Yaskawa INFORM job: A_ROOF_SIDE_0617_2_PAINT_58.JBI

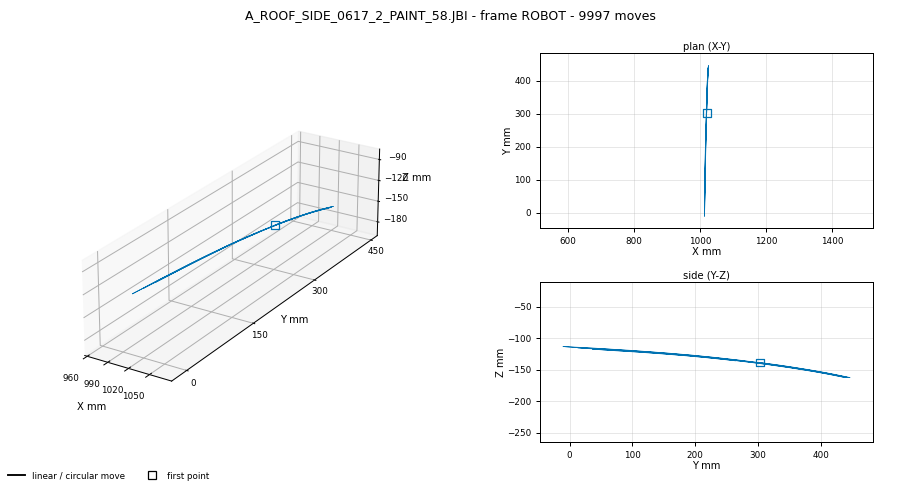
[picture p0: tool path of A_ROOF_SIDE_0617_2_PAINT_58.JBI in frame ROBOT, 9997 of 9997 moves have a stored position in this frame; points joined in program order, loops and branches not executed]
/JOB
//NAME A_ROOF_SIDE_0617_2_PAINT58
//POS
///NPOS 9997,0,0,0,0,0
///TOOL 1
///USER 0
///POSTYPE ROBOT
///RECTAN
///RCONF 1,0,0,0,0,0,0,0,0,0,0,0,0,0,0,0,0,0,0,0,0,0,0,0
C00000=1019.451,302.645,-138.347,170.187,50.132,159.718
C00001=1019.458,302.892,-138.379,170.193,50.128,159.718
C00002=1019.464,303.141,-138.411,170.199,50.124,159.718
C00003=1019.471,303.388,-138.443,170.204,50.121,159.718
C00004=1019.478,303.636,-138.476,170.209,50.117,159.718
C00005=1019.484,303.884,-138.508,170.215,50.113,159.718
C00006=1019.491,304.131,-138.540,170.220,50.110,159.718
C00007=1019.498,304.379,-138.573,170.227,50.106,159.719
C00008=1019.504,304.627,-138.604,170.232,50.103,159.719
C00009=1019.511,304.875,-138.637,170.237,50.099,159.719
C00010=1019.517,305.122,-138.670,170.243,50.095,159.719
C00011=1019.524,305.370,-138.701,170.248,50.092,159.719
C00012=1019.530,305.618,-138.734,170.255,50.088,159.719
C00013=1019.538,305.866,-138.767,170.260,50.085,159.719
C00014=1019.544,306.113,-138.799,170.265,50.082,159.719
C00015=1019.550,306.362,-138.831,170.271,50.077,159.719
C00016=1019.557,306.609,-138.864,170.276,50.074,159.719
C00017=1019.564,306.857,-138.897,170.283,50.070,159.720
C00018=1019.570,307.101,-138.929,170.288,50.067,159.720
C00019=1019.576,307.344,-138.960,170.293,50.064,159.720
C00020=1019.583,307.587,-138.992,170.299,50.060,159.720
C00021=1019.590,307.830,-139.025,170.305,50.057,159.720
C00022=1019.596,308.074,-139.056,170.310,50.053,159.720
C00023=1019.604,308.318,-139.089,170.316,50.050,159.720
C00024=1019.610,308.562,-139.121,170.322,50.046,159.720
C00025=1019.617,308.805,-139.152,170.327,50.043,159.721
C00026=1019.624,309.052,-139.185,170.333,50.039,159.721
C00027=1019.630,309.300,-139.217,170.338,50.036,159.721
C00028=1019.637,309.548,-139.250,170.345,50.033,159.721
C00029=1019.644,309.796,-139.283,170.350,50.029,159.721
C00030=1019.650,310.043,-139.315,170.356,50.026,159.721
C00031=1019.658,310.291,-139.349,170.362,50.023,159.722
C00032=1019.663,310.539,-139.382,170.367,50.020,159.722
C00033=1019.669,310.786,-139.415,170.373,50.016,159.722
C00034=1019.677,311.034,-139.449,170.379,50.013,159.722
C00035=1019.683,311.282,-139.482,170.384,50.010,159.722
C00036=1019.689,311.529,-139.515,170.391,50.007,159.723
C00037=1019.696,311.777,-139.549,170.396,50.004,159.723
C00038=1019.702,312.025,-139.582,170.402,50.000,159.723
C00039=1019.709,312.272,-139.615,170.408,49.997,159.723
C00040=1019.715,312.520,-139.648,170.414,49.994,159.723
C00041=1019.721,312.767,-139.682,170.419,49.991,159.724
C00042=1019.728,313.015,-139.715,170.425,49.988,159.724
C00043=1019.735,313.263,-139.749,170.431,49.984,159.724
C00044=1019.741,313.510,-139.782,170.437,49.981,159.724
C00045=1019.748,313.758,-139.816,170.443,49.978,159.724
C00046=1019.754,314.006,-139.849,170.448,49.976,159.725
C00047=1019.761,314.254,-139.883,170.455,49.972,159.725
C00048=1019.768,314.500,-139.916,170.460,49.969,159.725
C00049=1019.775,314.749,-139.949,170.466,49.967,159.726
C00050=1019.780,314.996,-139.983,170.472,49.963,159.726
C00051=1019.788,315.244,-140.017,170.478,49.960,159.726
C00052=1019.794,315.491,-140.050,170.484,49.957,159.726
C00053=1019.801,315.739,-140.084,170.490,49.954,159.727
C00054=1019.807,315.986,-140.118,170.495,49.951,159.727
C00055=1019.814,316.235,-140.151,170.502,49.948,159.727
C00056=1019.820,316.482,-140.184,170.507,49.945,159.727
C00057=1019.828,316.729,-140.218,170.514,49.941,159.728
C00058=1019.834,316.977,-140.252,170.519,49.939,159.728
C00059=1019.840,317.225,-140.285,170.526,49.936,159.728
C00060=1019.848,317.472,-140.319,170.532,49.933,159.729
C00061=1019.854,317.719,-140.352,170.537,49.930,159.729
C00062=1019.861,317.967,-140.387,170.544,49.927,159.729
C00063=1019.868,318.215,-140.421,170.549,49.924,159.729
C00064=1019.874,318.462,-140.454,170.556,49.921,159.730
C00065=1019.881,318.710,-140.487,170.561,49.918,159.730
C00066=1019.888,318.958,-140.522,170.568,49.915,159.730
C00067=1019.894,319.205,-140.555,170.574,49.912,159.731
C00068=1019.902,319.453,-140.589,170.580,49.909,159.731
C00069=1019.909,319.701,-140.623,170.586,49.907,159.731
C00070=1019.915,319.949,-140.657,170.591,49.903,159.731
C00071=1019.922,320.196,-140.691,170.598,49.900,159.732
C00072=1019.929,320.443,-140.725,170.603,49.898,159.732
C00073=1019.936,320.691,-140.759,170.610,49.895,159.732
C00074=1019.943,320.939,-140.793,170.616,49.892,159.733
C00075=1019.950,321.187,-140.827,170.622,49.889,159.733
C00076=1019.957,321.434,-140.860,170.628,49.886,159.733
C00077=1019.963,321.682,-140.894,170.635,49.883,159.734
C00078=1019.971,321.928,-140.928,170.640,49.881,159.734
C00079=1019.978,322.174,-140.962,170.647,49.878,159.734
C00080=1019.984,322.420,-140.996,170.653,49.875,159.735
C00081=1019.991,322.666,-141.030,170.659,49.872,159.735
C00082=1019.998,322.912,-141.064,170.665,49.869,159.735
C00083=1020.005,323.158,-141.098,170.672,49.866,159.736
C00084=1020.012,323.404,-141.132,170.677,49.864,159.736
C00085=1020.019,323.650,-141.165,170.684,49.861,159.736
C00086=1020.026,323.898,-141.200,170.690,49.858,159.737
C00087=1020.033,324.146,-141.234,170.696,49.855,159.737
C00088=1020.040,324.393,-141.268,170.702,49.853,159.737
C00089=1020.047,324.641,-141.303,170.709,49.850,159.738
C00090=1020.054,324.888,-141.336,170.715,49.848,159.738
C00091=1020.062,325.135,-141.371,170.721,49.845,159.739
C00092=1020.069,325.383,-141.405,170.727,49.842,159.739
C00093=1020.075,325.631,-141.439,170.734,49.839,159.739
C00094=1020.083,325.878,-141.474,170.739,49.836,159.740
C00095=1020.090,326.126,-141.508,170.746,49.834,159.740
C00096=1020.097,326.373,-141.542,170.753,49.831,159.741
C00097=1020.104,326.621,-141.576,170.758,49.828,159.741
C00098=1020.111,326.868,-141.612,170.766,49.826,159.741
C00099=1020.118,327.115,-141.646,170.771,49.823,159.742
C00100=1020.125,327.363,-141.681,170.778,49.821,159.742
C00101=1020.131,327.611,-141.716,170.784,49.818,159.743
C00102=1020.139,327.858,-141.750,170.791,49.815,159.743
C00103=1020.145,328.106,-141.785,170.797,49.813,159.744
C00104=1020.152,328.353,-141.820,170.803,49.810,159.744
C00105=1020.159,328.600,-141.855,170.809,49.808,159.744
C00106=1020.167,328.848,-141.890,170.816,49.806,159.745
C00107=1020.174,329.095,-141.925,170.822,49.803,159.745
C00108=1020.181,329.343,-141.960,170.829,49.801,159.746
C00109=1020.187,329.591,-141.995,170.835,49.798,159.746
C00110=1020.195,329.838,-142.029,170.842,49.796,159.747
C00111=1020.201,330.085,-142.064,170.848,49.794,159.747
C00112=1020.208,330.333,-142.099,170.854,49.791,159.748
C00113=1020.216,330.580,-142.134,170.860,49.789,159.748
C00114=1020.223,330.828,-142.169,170.867,49.786,159.748
C00115=1020.230,331.075,-142.205,170.873,49.784,159.749
C00116=1020.237,331.322,-142.240,170.880,49.782,159.750
C00117=1020.244,331.569,-142.274,170.887,49.779,159.750
C00118=1020.251,331.818,-142.310,170.893,49.777,159.750
C00119=1020.258,332.065,-142.345,170.900,49.774,159.751
C00120=1020.265,332.312,-142.380,170.906,49.772,159.751
C00121=1020.273,332.560,-142.415,170.913,49.770,159.752
C00122=1020.280,332.807,-142.450,170.919,49.767,159.752
C00123=1020.287,333.054,-142.486,170.925,49.765,159.753
C00124=1020.294,333.301,-142.521,170.932,49.763,159.753
C00125=1020.301,333.550,-142.557,170.939,49.761,159.754
C00126=1020.308,333.796,-142.592,170.946,49.758,159.755
C00127=1020.315,334.044,-142.627,170.952,49.756,159.755
C00128=1020.322,334.292,-142.663,170.959,49.754,159.756
C00129=1020.329,334.538,-142.699,170.965,49.752,159.756
C00130=1020.336,334.786,-142.734,170.972,49.750,159.757
C00131=1020.343,335.034,-142.769,170.979,49.747,159.757
C00132=1020.351,335.281,-142.805,170.985,49.745,159.758
C00133=1020.357,335.528,-142.840,170.992,49.743,159.758
C00134=1020.365,335.775,-142.877,170.998,49.741,159.759
C00135=1020.372,336.023,-142.912,171.005,49.739,159.759
C00136=1020.379,336.270,-142.948,171.012,49.736,159.760
C00137=1020.386,336.518,-142.983,171.018,49.734,159.760
C00138=1020.393,336.762,-143.018,171.025,49.733,159.761
C00139=1020.401,337.005,-143.054,171.031,49.731,159.762
C00140=1020.408,337.250,-143.089,171.038,49.728,159.762
C00141=1020.415,337.493,-143.125,171.044,49.726,159.763
C00142=1020.422,337.737,-143.159,171.051,49.724,159.763
C00143=1020.429,337.981,-143.194,171.058,49.723,159.764
C00144=1020.436,338.225,-143.230,171.065,49.720,159.765
C00145=1020.444,338.469,-143.265,171.072,49.718,159.765
C00146=1020.451,338.716,-143.301,171.078,49.716,159.766
C00147=1020.459,338.963,-143.337,171.085,49.714,159.766
C00148=1020.466,339.211,-143.372,171.092,49.712,159.767
C00149=1020.473,339.458,-143.408,171.098,49.710,159.768
C00150=1020.480,339.705,-143.445,171.106,49.708,159.768
C00151=1020.487,339.953,-143.481,171.113,49.706,159.769
C00152=1020.495,340.200,-143.517,171.119,49.704,159.770
C00153=1020.502,340.447,-143.553,171.126,49.702,159.770
C00154=1020.509,340.695,-143.590,171.132,49.701,159.771
C00155=1020.516,340.941,-143.626,171.139,49.698,159.771
C00156=1020.524,341.189,-143.662,171.147,49.697,159.772
C00157=1020.531,341.436,-143.698,171.153,49.695,159.773
C00158=1020.538,341.683,-143.735,171.160,49.693,159.773
C00159=1020.545,341.931,-143.771,171.167,49.691,159.774
C00160=1020.553,342.178,-143.807,171.175,49.689,159.775
C00161=1020.561,342.426,-143.843,171.181,49.687,159.775
C00162=1020.567,342.673,-143.880,171.188,49.685,159.776
C00163=1020.575,342.919,-143.917,171.195,49.684,159.777
C00164=1020.583,343.167,-143.953,171.201,49.682,159.777
C00165=1020.590,343.415,-143.990,171.209,49.680,159.778
C00166=1020.597,343.661,-144.026,171.216,49.678,159.779
C00167=1020.605,343.908,-144.063,171.223,49.677,159.780
C00168=1020.612,344.156,-144.099,171.230,49.674,159.780
C00169=1020.619,344.403,-144.136,171.237,49.673,159.781
C00170=1020.627,344.650,-144.173,171.244,49.671,159.782
C00171=1020.634,344.897,-144.209,171.251,49.670,159.782
C00172=1020.641,345.145,-144.245,171.258,49.668,159.783
C00173=1020.649,345.392,-144.282,171.265,49.666,159.784
C00174=1020.656,345.639,-144.319,171.273,49.664,159.784
C00175=1020.664,345.886,-144.356,171.279,49.662,159.785
C00176=1020.672,346.134,-144.392,171.286,49.661,159.786
C00177=1020.679,346.381,-144.430,171.294,49.659,159.787
C00178=1020.687,346.628,-144.466,171.301,49.657,159.787
C00179=1020.695,346.875,-144.503,171.308,49.656,159.788
C00180=1020.701,347.122,-144.539,171.315,49.654,159.789
C00181=1020.709,347.369,-144.576,171.322,49.653,159.790
C00182=1020.716,347.617,-144.613,171.330,49.651,159.790
C00183=1020.724,347.863,-144.650,171.337,49.649,159.791
C00184=1020.731,348.111,-144.687,171.344,49.648,159.792
C00185=1020.739,348.357,-144.724,171.351,49.646,159.793
C00186=1020.746,348.605,-144.761,171.358,49.644,159.793
C00187=1020.754,348.852,-144.799,171.366,49.643,159.794
C00188=1020.762,349.099,-144.836,171.374,49.642,159.795
C00189=1020.769,349.346,-144.873,171.380,49.640,159.796
C00190=1020.777,349.593,-144.910,171.387,49.638,159.797
C00191=1020.784,349.840,-144.948,171.395,49.637,159.797
C00192=1020.792,350.088,-144.986,171.402,49.636,159.798
C00193=1020.800,350.335,-145.022,171.410,49.634,159.799
C00194=1020.807,350.582,-145.060,171.416,49.633,159.800
C00195=1020.815,350.829,-145.097,171.424,49.631,159.801
C00196=1020.822,351.076,-145.134,171.431,49.630,159.802
C00197=1020.830,351.323,-145.172,171.439,49.628,159.802
C00198=1020.837,351.560,-145.207,171.447,49.627,159.803
C00199=1020.844,351.797,-145.243,171.453,49.626,159.804
C00200=1020.851,352.033,-145.279,171.460,49.624,159.805
C00201=1020.859,352.270,-145.315,171.467,49.623,159.806
C00202=1020.866,352.506,-145.351,171.474,49.621,159.806
C00203=1020.874,352.743,-145.386,171.482,49.620,159.807
C00204=1020.881,352.980,-145.423,171.489,49.619,159.808
C00205=1020.888,353.217,-145.459,171.496,49.618,159.809
C00206=1020.897,353.463,-145.497,171.504,49.616,159.810
C00207=1020.904,353.711,-145.534,171.511,49.615,159.811
C00208=1020.912,353.958,-145.572,171.519,49.613,159.812
C00209=1020.920,354.204,-145.609,171.526,49.613,159.813
C00210=1020.928,354.452,-145.647,171.533,49.611,159.813
C00211=1020.935,354.699,-145.685,171.541,49.610,159.814
C00212=1020.943,354.945,-145.723,171.549,49.609,159.815
C00213=1020.950,355.193,-145.761,171.556,49.608,159.816
C00214=1020.959,355.439,-145.799,171.564,49.606,159.817
C00215=1020.966,355.687,-145.836,171.571,49.605,159.818
C00216=1020.974,355.934,-145.875,171.579,49.604,159.819
C00217=1020.982,356.180,-145.913,171.587,49.603,159.820
C00218=1020.990,356.440,-145.952,171.595,49.601,159.821
C00219=1020.998,356.698,-145.992,171.602,49.600,159.822
C00220=1021.006,356.956,-146.031,171.611,49.599,159.823
C00221=1021.014,357.214,-146.072,171.619,49.598,159.824
C00222=1021.023,357.461,-146.110,171.626,49.596,159.825
C00223=1021.031,357.708,-146.148,171.634,49.595,159.826
C00224=1021.038,357.955,-146.186,171.642,49.594,159.827
C00225=1021.046,358.202,-146.224,171.650,49.593,159.827
C00226=1021.054,358.449,-146.263,171.657,49.592,159.828
C00227=1021.062,358.696,-146.301,171.665,49.591,159.829
C00228=1021.069,358.942,-146.340,171.673,49.590,159.830
C00229=1021.078,359.190,-146.378,171.681,49.589,159.832
C00230=1021.086,359.436,-146.416,171.689,49.588,159.833
C00231=1021.094,359.683,-146.454,171.697,49.587,159.833
C00232=1021.102,359.930,-146.493,171.704,49.586,159.834
C00233=1021.109,360.177,-146.532,171.712,49.585,159.835
C00234=1021.117,360.424,-146.570,171.720,49.584,159.836
C00235=1021.125,360.671,-146.609,171.728,49.583,159.838
C00236=1021.133,360.918,-146.647,171.736,49.582,159.839
C00237=1021.141,361.165,-146.686,171.743,49.581,159.839
C00238=1021.149,361.411,-146.725,171.752,49.580,159.841
C00239=1021.157,361.658,-146.764,171.760,49.579,159.842
C00240=1021.164,361.906,-146.803,171.768,49.578,159.843
C00241=1021.172,362.152,-146.842,171.776,49.577,159.844
C00242=1021.180,362.399,-146.880,171.784,49.576,159.845
C00243=1021.189,362.646,-146.919,171.792,49.576,159.846
C00244=1021.196,362.892,-146.958,171.800,49.575,159.847
C00245=1021.205,363.139,-146.996,171.808,49.574,159.848
C00246=1021.213,363.386,-147.036,171.816,49.573,159.849
C00247=1021.220,363.634,-147.075,171.824,49.573,159.850
C00248=1021.229,363.881,-147.114,171.833,49.571,159.851
C00249=1021.236,364.127,-147.153,171.841,49.571,159.852
C00250=1021.245,364.373,-147.192,171.848,49.570,159.853
C00251=1021.253,364.620,-147.230,171.857,49.569,159.855
C00252=1021.261,364.867,-147.270,171.865,49.569,159.856
C00253=1021.270,365.114,-147.308,171.872,49.567,159.857
C00254=1021.277,365.361,-147.348,171.882,49.567,159.858
C00255=1021.286,365.608,-147.388,171.890,49.566,159.859
C00256=1021.293,365.854,-147.426,171.897,49.565,159.860
C00257=1021.302,366.101,-147.465,171.906,49.565,159.861
C00258=1021.310,366.347,-147.505,171.914,49.564,159.862
C00259=1021.318,366.593,-147.544,171.923,49.563,159.864
C00260=1021.327,366.838,-147.583,171.931,49.563,159.865
C00261=1021.335,367.084,-147.622,171.939,49.562,159.866
C00262=1021.343,367.331,-147.661,171.947,49.561,159.867
C00263=1021.352,367.576,-147.701,171.956,49.560,159.868
C00264=1021.359,367.822,-147.739,171.964,49.560,159.869
C00265=1021.368,368.068,-147.779,171.972,49.559,159.871
C00266=1021.377,368.314,-147.819,171.980,49.559,159.872
C00267=1021.385,368.561,-147.858,171.989,49.558,159.873
C00268=1021.393,368.808,-147.898,171.997,49.557,159.874
C00269=1021.401,369.055,-147.937,172.006,49.557,159.875
C00270=1021.409,369.301,-147.977,172.014,49.556,159.877
C00271=1021.418,369.547,-148.017,172.023,49.556,159.878
C00272=1021.425,369.794,-148.057,172.031,49.556,159.879
C00273=1021.434,370.041,-148.097,172.039,49.555,159.880
C00274=1021.442,370.288,-148.137,172.049,49.554,159.882
C00275=1021.451,370.535,-148.177,172.057,49.554,159.883
C00276=1021.459,370.781,-148.217,172.065,49.554,159.884
C00277=1021.467,371.028,-148.256,172.074,49.553,159.885
C00278=1021.475,371.274,-148.297,172.082,49.553,159.887
C00279=1021.484,371.521,-148.336,172.091,49.553,159.888
C00280=1021.492,371.768,-148.377,172.100,49.552,159.889
C00281=1021.501,372.014,-148.416,172.108,49.551,159.890
C00282=1021.509,372.261,-148.457,172.117,49.551,159.892
C00283=1021.518,372.508,-148.497,172.126,49.551,159.893
C00284=1021.526,372.754,-148.537,172.134,49.551,159.894
C00285=1021.535,373.000,-148.577,172.143,49.550,159.896
C00286=1021.543,373.248,-148.618,172.152,49.550,159.897
C00287=1021.552,373.494,-148.658,172.161,49.549,159.898
C00288=1021.560,373.740,-148.698,172.169,49.549,159.900
C00289=1021.569,373.987,-148.738,172.178,49.549,159.901
C00290=1021.577,374.234,-148.779,172.187,49.548,159.902
C00291=1021.586,374.480,-148.819,172.196,49.549,159.904
C00292=1021.594,374.727,-148.860,172.205,49.548,159.905
C00293=1021.603,374.973,-148.900,172.213,49.548,159.906
C00294=1021.611,375.220,-148.940,172.223,49.548,159.908
C00295=1021.620,375.466,-148.980,172.231,49.547,159.909
C00296=1021.629,375.713,-149.021,172.240,49.547,159.910
C00297=1021.637,375.959,-149.061,172.249,49.547,159.912
C00298=1021.646,376.206,-149.102,172.258,49.547,159.913
C00299=1021.655,376.453,-149.143,172.268,49.546,159.915
C00300=1021.664,376.699,-149.184,172.276,49.546,159.916
C00301=1021.672,376.946,-149.225,172.286,49.546,159.917
C00302=1021.680,377.192,-149.266,172.294,49.546,159.919
C00303=1021.689,377.439,-149.307,172.304,49.546,159.920
C00304=1021.697,377.684,-149.348,172.312,49.546,159.922
C00305=1021.707,377.931,-149.388,172.322,49.546,159.923
C00306=1021.715,378.177,-149.429,172.330,49.546,159.924
C00307=1021.724,378.424,-149.471,172.340,49.546,159.926
C00308=1021.732,378.671,-149.512,172.349,49.545,159.927
C00309=1021.741,378.916,-149.553,172.358,49.545,159.929
C00310=1021.749,379.163,-149.594,172.367,49.545,159.930
C00311=1021.759,379.409,-149.635,172.376,49.546,159.932
C00312=1021.768,379.656,-149.676,172.385,49.546,159.933
C00313=1021.776,379.902,-149.718,172.395,49.545,159.935
C00314=1021.785,380.149,-149.759,172.404,49.546,159.936
C00315=1021.793,380.395,-149.800,172.413,49.546,159.938
C00316=1021.802,380.642,-149.841,172.423,49.546,159.939
C00317=1021.811,380.888,-149.882,172.432,49.546,159.941
C00318=1021.821,381.155,-149.928,172.442,49.546,159.942
C00319=1021.831,381.422,-149.972,172.452,49.546,159.944
C00320=1021.840,381.689,-150.017,172.463,49.546,159.946
C00321=1021.849,381.956,-150.062,172.473,49.546,159.947
C00322=1021.858,382.202,-150.103,172.482,49.546,159.949
C00323=1021.867,382.449,-150.145,172.492,49.546,159.950
C00324=1021.877,382.695,-150.186,172.501,49.547,159.952
C00325=1021.886,382.941,-150.228,172.510,49.547,159.953
C00326=1021.895,383.188,-150.270,172.520,49.547,159.955
C00327=1021.904,383.434,-150.311,172.530,49.547,159.957
C00328=1021.913,383.680,-150.353,172.540,49.547,159.958
C00329=1021.921,383.927,-150.395,172.548,49.548,159.960
C00330=1021.931,384.173,-150.436,172.558,49.548,159.961
C00331=1021.940,384.419,-150.478,172.568,49.548,159.963
C00332=1021.949,384.665,-150.519,172.578,49.548,159.965
C00333=1021.959,384.912,-150.561,172.587,49.548,159.966
C00334=1021.968,385.158,-150.604,172.597,49.549,159.968
C00335=1021.977,385.405,-150.646,172.607,49.549,159.970
C00336=1021.986,385.651,-150.687,172.617,49.549,159.971
C00337=1021.995,385.897,-150.730,172.626,49.550,159.973
C00338=1022.004,386.143,-150.771,172.636,49.550,159.974
C00339=1022.013,386.390,-150.814,172.646,49.551,159.976
C00340=1022.023,386.636,-150.856,172.655,49.551,159.978
C00341=1022.032,386.882,-150.898,172.665,49.551,159.979
C00342=1022.041,387.128,-150.940,172.675,49.552,159.981
C00343=1022.050,387.374,-150.983,172.685,49.552,159.983
C00344=1022.060,387.621,-151.025,172.695,49.552,159.984
C00345=1022.069,387.867,-151.067,172.705,49.553,159.986
C00346=1022.077,388.113,-151.110,172.715,49.553,159.988
C00347=1022.087,388.360,-151.152,172.725,49.554,159.990
C00348=1022.096,388.605,-151.195,172.735,49.555,159.991
C00349=1022.105,388.851,-151.237,172.745,49.555,159.993
C00350=1022.115,389.098,-151.280,172.755,49.555,159.995
C00351=1022.124,389.344,-151.323,172.765,49.556,159.997
C00352=1022.133,389.589,-151.365,172.775,49.557,159.998
C00353=1022.143,389.836,-151.408,172.785,49.557,160.000
C00354=1022.152,390.082,-151.451,172.796,49.557,160.002
C00355=1022.161,390.328,-151.494,172.806,49.558,160.004
C00356=1022.170,390.574,-151.536,172.816,49.559,160.005
C00357=1022.180,390.820,-151.579,172.826,49.559,160.007
C00358=1022.189,391.066,-151.622,172.836,49.560,160.009
C00359=1022.199,391.312,-151.666,172.846,49.561,160.011
C00360=1022.208,391.558,-151.708,172.856,49.561,160.013
C00361=1022.218,391.805,-151.751,172.868,49.562,160.015
C00362=1022.227,392.050,-151.793,172.878,49.563,160.017
C00363=1022.237,392.296,-151.837,172.888,49.563,160.018
C00364=1022.246,392.542,-151.880,172.898,49.564,160.020
C00365=1022.256,392.789,-151.923,172.908,49.565,160.022
C00366=1022.265,393.035,-151.967,172.919,49.565,160.024
C00367=1022.274,393.280,-152.009,172.930,49.566,160.026
C00368=1022.284,393.526,-152.053,172.940,49.567,160.028
C00369=1022.294,393.772,-152.097,172.950,49.568,160.030
C00370=1022.303,394.018,-152.139,172.961,49.569,160.031
C00371=1022.312,394.264,-152.183,172.972,49.570,160.033
C00372=1022.323,394.510,-152.227,172.982,49.570,160.035
C00373=1022.332,394.757,-152.270,172.993,49.572,160.037
C00374=1022.341,395.002,-152.313,173.004,49.572,160.039
C00375=1022.351,395.248,-152.357,173.014,49.573,160.041
C00376=1022.361,395.494,-152.401,173.025,49.574,160.043
C00377=1022.371,395.740,-152.445,173.036,49.575,160.045
C00378=1022.382,396.044,-152.499,173.048,49.576,160.047
C00379=1022.395,396.348,-152.553,173.062,49.577,160.050
C00380=1022.407,396.652,-152.607,173.075,49.578,160.052
C00381=1022.419,396.956,-152.661,173.089,49.579,160.055
C00382=1022.429,397.203,-152.705,173.100,49.581,160.057
C00383=1022.439,397.448,-152.748,173.111,49.581,160.059
C00384=1022.448,397.694,-152.793,173.122,49.583,160.061
C00385=1022.459,397.940,-152.837,173.133,49.583,160.063
C00386=1022.468,398.186,-152.881,173.143,49.585,160.065
C00387=1022.478,398.432,-152.924,173.155,49.586,160.067
C00388=1022.488,398.677,-152.969,173.165,49.587,160.069
C00389=1022.497,398.923,-153.013,173.177,49.588,160.071
C00390=1022.508,399.168,-153.057,173.188,49.589,160.073
C00391=1022.517,399.415,-153.102,173.199,49.590,160.075
C00392=1022.527,399.660,-153.146,173.209,49.591,160.077
C00393=1022.537,399.906,-153.190,173.221,49.592,160.079
C00394=1022.547,400.152,-153.235,173.233,49.593,160.082
C00395=1022.557,400.398,-153.280,173.243,49.595,160.084
C00396=1022.567,400.644,-153.323,173.255,49.596,160.086
C00397=1022.577,400.889,-153.368,173.266,49.597,160.088
C00398=1022.587,401.135,-153.413,173.277,49.598,160.090
C00399=1022.597,401.381,-153.458,173.289,49.600,160.092
C00400=1022.607,401.626,-153.502,173.301,49.601,160.095
C00401=1022.617,401.871,-153.547,173.311,49.602,160.097
C00402=1022.627,402.118,-153.592,173.323,49.603,160.099
C00403=1022.637,402.363,-153.637,173.334,49.604,160.101
C00404=1022.647,402.609,-153.682,173.346,49.606,160.103
C00405=1022.657,402.855,-153.727,173.357,49.608,160.106
C00406=1022.668,403.100,-153.772,173.369,49.609,160.108
C00407=1022.677,403.346,-153.816,173.380,49.610,160.110
C00408=1022.688,403.592,-153.862,173.392,49.611,160.112
C00409=1022.697,403.837,-153.906,173.404,49.613,160.115
C00410=1022.708,404.083,-153.952,173.415,49.614,160.117
C00411=1022.718,404.328,-153.997,173.427,49.616,160.119
C00412=1022.728,404.575,-154.042,173.439,49.618,160.121
C00413=1022.739,404.819,-154.087,173.450,49.619,160.124
C00414=1022.749,405.065,-154.132,173.462,49.620,160.126
C00415=1022.760,405.311,-154.178,173.474,49.622,160.128
C00416=1022.769,405.557,-154.223,173.486,49.623,160.130
C00417=1022.780,405.802,-154.269,173.498,49.625,160.133
C00418=1022.790,406.048,-154.314,173.510,49.626,160.135
C00419=1022.800,406.293,-154.360,173.522,49.628,160.138
C00420=1022.812,406.539,-154.405,173.534,49.629,160.140
C00421=1022.822,406.785,-154.450,173.546,49.631,160.142
C00422=1022.833,407.030,-154.496,173.558,49.633,160.145
C00423=1022.843,407.276,-154.542,173.570,49.634,160.147
C00424=1022.853,407.521,-154.588,173.582,49.636,160.150
C00425=1022.864,407.767,-154.633,173.594,49.637,160.152
C00426=1022.874,408.013,-154.679,173.607,49.639,160.154
C00427=1022.886,408.258,-154.724,173.619,49.640,160.157
C00428=1022.896,408.504,-154.770,173.631,49.642,160.159
C00429=1022.907,408.749,-154.816,173.643,49.643,160.161
C00430=1022.918,408.995,-154.862,173.655,49.646,160.164
C00431=1022.928,409.240,-154.908,173.667,49.647,160.166
C00432=1022.939,409.486,-154.954,173.680,49.648,160.169
C00433=1022.950,409.731,-155.000,173.692,49.651,160.171
C00434=1022.960,409.976,-155.046,173.704,49.652,160.174
C00435=1022.970,410.222,-155.093,173.717,49.654,160.176
C00436=1022.981,410.467,-155.139,173.729,49.655,160.179
C00437=1022.992,410.713,-155.185,173.742,49.658,160.181
C00438=1023.007,411.039,-155.247,173.758,49.661,160.185
C00439=1023.021,411.366,-155.309,173.775,49.662,160.188
C00440=1023.035,411.692,-155.371,173.792,49.665,160.192
C00441=1023.049,412.019,-155.432,173.809,49.668,160.195
C00442=1023.060,412.264,-155.479,173.821,49.669,160.198
C00443=1023.072,412.510,-155.526,173.835,49.671,160.200
C00444=1023.082,412.755,-155.573,173.847,49.673,160.203
C00445=1023.093,413.000,-155.620,173.860,49.675,160.206
C00446=1023.104,413.246,-155.666,173.873,49.677,160.208
C00447=1023.115,413.491,-155.713,173.886,49.679,160.211
C00448=1023.126,413.736,-155.759,173.899,49.682,160.214
C00449=1023.138,413.982,-155.806,173.912,49.683,160.216
C00450=1023.148,414.227,-155.854,173.925,49.686,160.219
C00451=1023.159,414.473,-155.901,173.938,49.687,160.222
C00452=1023.170,414.718,-155.947,173.951,49.689,160.224
C00453=1023.182,414.963,-155.995,173.964,49.692,160.227
C00454=1023.193,415.208,-156.042,173.977,49.693,160.230
C00455=1023.204,415.454,-156.089,173.991,49.696,160.233
C00456=1023.215,415.700,-156.136,174.004,49.698,160.235
C00457=1023.227,415.944,-156.184,174.017,49.700,160.238
C00458=1023.237,416.190,-156.231,174.031,49.702,160.241
C00459=1023.249,416.435,-156.279,174.044,49.704,160.244
C00460=1023.259,416.680,-156.326,174.057,49.707,160.246
C00461=1023.271,416.925,-156.374,174.070,49.709,160.249
C00462=1023.282,417.171,-156.422,174.084,49.711,160.252
C00463=1023.293,417.416,-156.469,174.098,49.713,160.255
C00464=1023.304,417.661,-156.517,174.112,49.716,160.258
C00465=1023.316,417.906,-156.565,174.125,49.718,160.261
C00466=1023.327,418.152,-156.613,174.138,49.721,160.264
C00467=1023.339,418.397,-156.661,174.152,49.723,160.266
C00468=1023.351,418.642,-156.708,174.166,49.725,160.269
C00469=1023.361,418.886,-156.756,174.179,49.727,160.272
C00470=1023.373,419.131,-156.804,174.193,49.730,160.275
C00471=1023.384,419.377,-156.852,174.207,49.732,160.278
C00472=1023.396,419.622,-156.900,174.221,49.734,160.281
C00473=1023.407,419.867,-156.948,174.235,49.737,160.284
C00474=1023.419,420.112,-156.996,174.249,49.739,160.287
C00475=1023.431,420.358,-157.045,174.263,49.741,160.290
C00476=1023.443,420.603,-157.093,174.277,49.744,160.293
C00477=1023.455,420.848,-157.141,174.291,49.746,160.296
C00478=1023.466,421.093,-157.189,174.305,49.749,160.299
C00479=1023.478,421.338,-157.237,174.319,49.751,160.302
C00480=1023.490,421.584,-157.286,174.334,49.754,160.305
C00481=1023.502,421.828,-157.335,174.348,49.756,160.308
C00482=1023.513,422.073,-157.383,174.362,49.759,160.311
C00483=1023.524,422.318,-157.432,174.376,49.762,160.314
C00484=1023.537,422.563,-157.481,174.391,49.764,160.317
C00485=1023.549,422.808,-157.530,174.405,49.767,160.320
C00486=1023.560,423.053,-157.578,174.420,49.770,160.324
C00487=1023.572,423.299,-157.627,174.435,49.772,160.327
C00488=1023.584,423.543,-157.676,174.449,49.775,160.330
C00489=1023.595,423.788,-157.725,174.464,49.777,160.333
C00490=1023.608,424.033,-157.774,174.478,49.780,160.336
C00491=1023.619,424.278,-157.823,174.493,49.782,160.339
C00492=1023.632,424.523,-157.873,174.507,49.785,160.342
C00493=1023.644,424.767,-157.921,174.523,49.788,160.346
C00494=1023.656,425.013,-157.970,174.537,49.791,160.349
C00495=1023.668,425.258,-158.020,174.552,49.793,160.352
C00496=1023.679,425.503,-158.069,174.568,49.796,160.355
C00497=1023.692,425.747,-158.118,174.582,49.799,160.359
C00498=1023.709,426.085,-158.187,174.603,49.803,160.363
C00499=1023.725,426.423,-158.256,174.624,49.807,160.368
C00500=1023.742,426.762,-158.324,174.644,49.811,160.372
C00501=1023.758,427.099,-158.392,174.665,49.815,160.377
C00502=1023.771,427.344,-158.442,174.681,49.818,160.380
C00503=1023.783,427.589,-158.492,174.696,49.821,160.384
C00504=1023.796,427.833,-158.542,174.712,49.824,160.387
C00505=1023.808,428.078,-158.592,174.727,49.827,160.391
C00506=1023.821,428.323,-158.642,174.743,49.830,160.394
C00507=1023.833,428.568,-158.692,174.758,49.833,160.397
C00508=1023.845,428.812,-158.742,174.774,49.836,160.401
C00509=1023.857,429.057,-158.792,174.789,49.839,160.404
C00510=1023.869,429.301,-158.842,174.805,49.841,160.408
C00511=1023.882,429.546,-158.893,174.821,49.845,160.411
C00512=1023.895,429.791,-158.943,174.836,49.848,160.415
C00513=1023.908,430.036,-158.993,174.852,49.851,160.418
C00514=1023.920,430.280,-159.044,174.868,49.854,160.422
C00515=1023.933,430.525,-159.094,174.883,49.858,160.425
C00516=1023.945,430.769,-159.145,174.899,49.860,160.429
C00517=1023.958,431.014,-159.195,174.916,49.864,160.433
C00518=1023.971,431.259,-159.246,174.932,49.867,160.436
C00519=1023.983,431.503,-159.296,174.948,49.870,160.440
C00520=1023.996,431.748,-159.347,174.964,49.873,160.443
C00521=1024.009,431.991,-159.397,174.980,49.876,160.447
C00522=1024.022,432.236,-159.448,174.996,49.880,160.451
C00523=1024.035,432.481,-159.499,175.013,49.883,160.454
C00524=1024.048,432.726,-159.549,175.029,49.886,160.458
C00525=1024.061,432.970,-159.601,175.046,49.889,160.462
C00526=1024.074,433.215,-159.652,175.062,49.893,160.465
C00527=1024.087,433.459,-159.703,175.079,49.896,160.469
C00528=1024.100,433.704,-159.754,175.095,49.899,160.473
C00529=1024.112,433.948,-159.805,175.112,49.903,160.477
C00530=1024.125,434.193,-159.857,175.128,49.906,160.480
C00531=1024.138,434.437,-159.909,175.145,49.910,160.484
C00532=1024.151,434.681,-159.960,175.162,49.913,160.488
C00533=1024.165,434.926,-160.011,175.178,49.917,160.492
C00534=1024.178,435.169,-160.063,175.196,49.920,160.496
C00535=1024.191,435.414,-160.115,175.213,49.923,160.499
C00536=1024.204,435.659,-160.166,175.230,49.927,160.503
C00537=1024.218,435.903,-160.218,175.247,49.930,160.507
C00538=1024.230,436.147,-160.270,175.264,49.934,160.511
C00539=1024.244,436.391,-160.322,175.281,49.938,160.515
C00540=1024.257,436.635,-160.374,175.298,49.941,160.519
C00541=1024.271,436.880,-160.426,175.315,49.945,160.523
C00542=1024.284,437.124,-160.478,175.333,49.949,160.527
C00543=1024.298,437.368,-160.529,175.350,49.952,160.531
C00544=1024.311,437.613,-160.581,175.368,49.956,160.535
C00545=1024.324,437.857,-160.634,175.386,49.959,160.539
C00546=1024.338,438.101,-160.686,175.404,49.963,160.543
C00547=1024.351,438.345,-160.738,175.421,49.967,160.547
C00548=1024.365,438.589,-160.791,175.439,49.970,160.551
C00549=1024.378,438.833,-160.843,175.456,49.974,160.555
C00550=1024.392,439.077,-160.896,175.475,49.978,160.560
C00551=1024.406,439.322,-160.948,175.493,49.982,160.564
C00552=1024.420,439.566,-161.001,175.510,49.985,160.568
C00553=1024.433,439.810,-161.054,175.529,49.989,160.572
C00554=1024.447,440.053,-161.107,175.546,49.993,160.576
C00555=1024.461,440.298,-161.160,175.565,49.997,160.581
C00556=1024.475,440.541,-161.212,175.583,50.001,160.585
C00557=1024.488,440.785,-161.265,175.602,50.004,160.589
C00558=1024.511,441.179,-161.351,175.631,50.011,160.596
C00559=1024.533,441.573,-161.436,175.660,50.017,160.603
C00560=1024.556,441.966,-161.521,175.691,50.023,160.610
C00561=1024.580,442.360,-161.608,175.721,50.030,160.617
C00562=1024.594,442.603,-161.660,175.739,50.034,160.621
C00563=1024.609,442.846,-161.712,175.759,50.038,160.625
C00564=1024.625,443.089,-161.764,175.777,50.041,160.630
C00565=1024.641,443.334,-161.815,175.797,50.044,160.634
C00566=1024.657,443.577,-161.866,175.816,50.048,160.638
C00567=1024.673,443.820,-161.917,175.835,50.052,160.643
C00568=1024.691,444.064,-161.968,175.855,50.055,160.647
C00569=1024.709,444.309,-162.018,175.873,50.059,160.651
C00570=1024.726,444.552,-162.067,175.893,50.062,160.656
C00571=1024.746,444.796,-162.116,175.912,50.065,160.660
C00572=1024.765,445.040,-162.165,175.932,50.068,160.664
C00573=1024.784,445.285,-162.214,175.952,50.072,160.669
C00574=1024.805,445.529,-162.261,175.972,50.075,160.673
C00575=1024.824,445.773,-162.309,175.991,50.078,160.677
C00576=1024.845,446.017,-162.356,176.012,50.080,160.681
C00577=1024.867,446.262,-162.403,176.032,50.083,160.686
C00578=1024.405,444.052,-162.296,175.845,50.118,160.665
C00579=1024.388,443.808,-162.246,175.826,50.114,160.660
C00580=1024.371,443.564,-162.196,175.807,50.111,160.656
C00581=1024.355,443.320,-162.145,175.788,50.108,160.652
C00582=1024.339,443.077,-162.093,175.769,50.104,160.648
C00583=1024.318,442.749,-162.024,175.743,50.099,160.642
C00584=1024.298,442.421,-161.953,175.718,50.094,160.636
C00585=1024.279,442.095,-161.882,175.693,50.090,160.630
C00586=1024.259,441.768,-161.811,175.668,50.084,160.624
C00587=1024.247,441.550,-161.764,175.651,50.080,160.620
C00588=1024.235,441.332,-161.716,175.634,50.078,160.617
C00589=1024.222,441.115,-161.669,175.618,50.074,160.613
C00590=1024.209,440.897,-161.622,175.602,50.070,160.609
C00591=1024.196,440.653,-161.569,175.583,50.067,160.605
C00592=1024.182,440.409,-161.516,175.565,50.063,160.601
C00593=1024.168,440.165,-161.463,175.547,50.059,160.596
C00594=1024.154,439.921,-161.410,175.528,50.056,160.592
C00595=1024.140,439.677,-161.358,175.511,50.052,160.588
C00596=1024.127,439.433,-161.306,175.493,50.048,160.584
C00597=1024.113,439.188,-161.252,175.474,50.045,160.580
C00598=1024.099,438.945,-161.199,175.456,50.041,160.576
C00599=1024.086,438.701,-161.148,175.438,50.038,160.572
C00600=1024.072,438.457,-161.095,175.420,50.034,160.567
C00601=1024.059,438.212,-161.042,175.403,50.030,160.563
C00602=1024.045,437.969,-160.990,175.385,50.026,160.559
C00603=1024.032,437.724,-160.938,175.368,50.023,160.555
C00604=1024.018,437.480,-160.886,175.350,50.020,160.551
C00605=1024.005,437.236,-160.834,175.332,50.016,160.547
C00606=1023.991,436.991,-160.782,175.315,50.012,160.543
C00607=1023.978,436.747,-160.730,175.297,50.009,160.539
C00608=1023.965,436.503,-160.678,175.280,50.005,160.535
C00609=1023.951,436.258,-160.626,175.263,50.002,160.531
C00610=1023.938,436.014,-160.574,175.246,49.999,160.528
C00611=1023.925,435.770,-160.523,175.229,49.995,160.524
C00612=1023.911,435.526,-160.471,175.211,49.992,160.520
C00613=1023.898,435.281,-160.420,175.194,49.988,160.516
C00614=1023.885,435.037,-160.367,175.178,49.985,160.512
C00615=1023.872,434.793,-160.316,175.161,49.981,160.508
C00616=1023.859,434.548,-160.264,175.144,49.979,160.504
C00617=1023.846,434.303,-160.213,175.126,49.975,160.501
C00618=1023.833,434.060,-160.162,175.111,49.972,160.497
C00619=1023.820,433.815,-160.110,175.093,49.968,160.493
C00620=1023.807,433.571,-160.060,175.076,49.965,160.489
C00621=1023.794,433.326,-160.008,175.060,49.962,160.486
C00622=1023.781,433.082,-159.957,175.043,49.959,160.482
C00623=1023.768,432.837,-159.906,175.028,49.955,160.478
C00624=1023.755,432.593,-159.855,175.011,49.952,160.474
C00625=1023.742,432.348,-159.804,174.995,49.949,160.471
C00626=1023.729,432.104,-159.753,174.978,49.946,160.467
C00627=1023.717,431.858,-159.702,174.962,49.943,160.463
C00628=1023.704,431.614,-159.652,174.945,49.940,160.460
C00629=1023.691,431.370,-159.601,174.929,49.937,160.456
C00630=1023.679,431.125,-159.551,174.913,49.933,160.453
C00631=1023.665,430.881,-159.500,174.897,49.930,160.449
C00632=1023.652,430.636,-159.449,174.881,49.927,160.446
C00633=1023.640,430.392,-159.399,174.865,49.924,160.442
C00634=1023.628,430.147,-159.349,174.849,49.922,160.438
C00635=1023.615,429.903,-159.298,174.833,49.919,160.435
C00636=1023.603,429.658,-159.248,174.817,49.915,160.431
C00637=1023.591,429.413,-159.198,174.802,49.912,160.428
C00638=1023.577,429.169,-159.148,174.786,49.909,160.424
C00639=1023.565,428.924,-159.098,174.771,49.907,160.421
C00640=1023.553,428.679,-159.048,174.755,49.904,160.418
C00641=1023.540,428.435,-158.998,174.739,49.901,160.414
C00642=1023.528,428.190,-158.948,174.724,49.898,160.411
C00643=1023.516,427.945,-158.898,174.708,49.895,160.407
C00644=1023.503,427.700,-158.847,174.693,49.892,160.404
C00645=1023.491,427.455,-158.797,174.677,49.889,160.401
C00646=1023.478,427.211,-158.748,174.662,49.886,160.397
C00647=1023.461,426.871,-158.679,174.641,49.883,160.393
C00648=1023.445,426.530,-158.609,174.620,49.879,160.388
C00649=1023.429,426.190,-158.541,174.599,49.875,160.383
C00650=1023.411,425.850,-158.471,174.578,49.871,160.379
C00651=1023.400,425.605,-158.422,174.562,49.868,160.375
C00652=1023.387,425.360,-158.373,174.548,49.865,160.372
C00653=1023.375,425.115,-158.324,174.532,49.862,160.369
C00654=1023.364,424.870,-158.275,174.517,49.860,160.366
C00655=1023.351,424.625,-158.226,174.503,49.857,160.363
C00656=1023.339,424.380,-158.177,174.488,49.855,160.359
C00657=1023.327,424.135,-158.127,174.474,49.852,160.356
C00658=1023.315,423.891,-158.078,174.459,49.850,160.353
C00659=1023.303,423.646,-158.029,174.444,49.847,160.350
C00660=1023.291,423.401,-157.980,174.429,49.845,160.347
C00661=1023.279,423.155,-157.932,174.414,49.842,160.343
C00662=1023.268,422.910,-157.883,174.400,49.839,160.340
C00663=1023.256,422.666,-157.834,174.386,49.837,160.337
C00664=1023.244,422.421,-157.785,174.371,49.835,160.334
C00665=1023.232,422.176,-157.736,174.357,49.832,160.331
C00666=1023.220,421.931,-157.688,174.343,49.829,160.328
C00667=1023.209,421.686,-157.639,174.328,49.827,160.325
C00668=1023.198,421.441,-157.591,174.314,49.825,160.322
C00669=1023.185,421.195,-157.542,174.300,49.822,160.319
C00670=1023.174,420.950,-157.494,174.285,49.820,160.316
C00671=1023.162,420.705,-157.446,174.271,49.818,160.313
C00672=1023.150,420.461,-157.398,174.257,49.815,160.310
C00673=1023.139,420.215,-157.349,174.243,49.813,160.307
C00674=1023.127,419.970,-157.302,174.230,49.810,160.304
C00675=1023.116,419.725,-157.253,174.215,49.808,160.301
C00676=1023.104,419.480,-157.206,174.201,49.806,160.298
C00677=1023.093,419.235,-157.157,174.187,49.804,160.295
C00678=1023.081,418.990,-157.109,174.174,49.802,160.292
C00679=1023.069,418.745,-157.061,174.160,49.799,160.289
C00680=1023.058,418.499,-157.013,174.146,49.797,160.287
C00681=1023.046,418.254,-156.966,174.132,49.795,160.284
C00682=1023.035,418.008,-156.918,174.119,49.793,160.281
C00683=1023.023,417.763,-156.870,174.105,49.790,160.278
C00684=1023.013,417.519,-156.822,174.091,49.788,160.275
C00685=1023.001,417.274,-156.774,174.077,49.786,160.272
C00686=1022.990,417.028,-156.727,174.064,49.784,160.269
C00687=1022.979,416.783,-156.679,174.050,49.782,160.266
C00688=1022.968,416.538,-156.633,174.038,49.779,160.264
C00689=1022.956,416.292,-156.584,174.024,49.777,160.261
C00690=1022.945,416.047,-156.537,174.010,49.775,160.258
C00691=1022.934,415.802,-156.489,173.997,49.773,160.255
C00692=1022.923,415.556,-156.442,173.983,49.771,160.252
C00693=1022.912,415.312,-156.395,173.971,49.769,160.250
C00694=1022.901,415.066,-156.347,173.958,49.767,160.247
C00695=1022.889,414.820,-156.300,173.944,49.765,160.244
C00696=1022.878,414.575,-156.254,173.931,49.763,160.242
C00697=1022.867,414.330,-156.207,173.918,49.761,160.239
C00698=1022.856,414.085,-156.160,173.905,49.759,160.236
C00699=1022.845,413.839,-156.113,173.892,49.757,160.234
C00700=1022.834,413.594,-156.066,173.879,49.755,160.231
C00701=1022.823,413.349,-156.019,173.866,49.754,160.228
C00702=1022.812,413.103,-155.972,173.853,49.752,160.226
C00703=1022.801,412.858,-155.926,173.840,49.750,160.223
C00704=1022.790,412.613,-155.879,173.827,49.748,160.220
C00705=1022.779,412.367,-155.832,173.814,49.746,160.218
C00706=1022.769,412.122,-155.786,173.802,49.744,160.215
C00707=1022.754,411.793,-155.723,173.785,49.742,160.212
C00708=1022.739,411.464,-155.661,173.767,49.739,160.208
C00709=1022.725,411.135,-155.599,173.751,49.737,160.205
C00710=1022.711,410.806,-155.536,173.733,49.735,160.201
C00711=1022.700,410.561,-155.490,173.721,49.733,160.199
C00712=1022.689,410.315,-155.443,173.708,49.731,160.196
C00713=1022.678,410.070,-155.397,173.696,49.730,160.194
C00714=1022.667,409.824,-155.351,173.684,49.728,160.191
C00715=1022.657,409.579,-155.305,173.671,49.726,160.189
C00716=1022.647,409.333,-155.258,173.659,49.725,160.187
C00717=1022.636,409.088,-155.212,173.646,49.723,160.184
C00718=1022.625,408.842,-155.167,173.634,49.721,160.182
C00719=1022.614,408.597,-155.121,173.621,49.720,160.179
C00720=1022.603,408.351,-155.075,173.609,49.718,160.177
C00721=1022.593,408.105,-155.029,173.597,49.717,160.174
C00722=1022.582,407.860,-154.984,173.585,49.715,160.172
C00723=1022.572,407.615,-154.938,173.572,49.714,160.170
C00724=1022.562,407.369,-154.893,173.560,49.712,160.167
C00725=1022.550,407.124,-154.847,173.548,49.711,160.165
C00726=1022.540,406.878,-154.802,173.536,49.709,160.162
C00727=1022.529,406.632,-154.756,173.524,49.707,160.160
C00728=1022.520,406.387,-154.711,173.513,49.706,160.158
C00729=1022.509,406.141,-154.665,173.501,49.705,160.155
C00730=1022.499,405.895,-154.620,173.489,49.703,160.153
C00731=1022.488,405.649,-154.574,173.477,49.702,160.151
C00732=1022.478,405.404,-154.530,173.464,49.701,160.148
C00733=1022.467,405.159,-154.484,173.452,49.699,160.146
C00734=1022.457,404.913,-154.439,173.441,49.698,160.144
C00735=1022.447,404.667,-154.393,173.430,49.696,160.142
C00736=1022.436,404.421,-154.348,173.418,49.695,160.139
C00737=1022.427,404.176,-154.303,173.406,49.694,160.137
C00738=1022.415,403.930,-154.258,173.394,49.693,160.135
C00739=1022.405,403.685,-154.213,173.382,49.691,160.132
C00740=1022.396,403.439,-154.168,173.371,49.690,160.130
C00741=1022.385,403.193,-154.123,173.359,49.688,160.128
C00742=1022.375,402.948,-154.077,173.347,49.687,160.126
C00743=1022.365,402.702,-154.032,173.336,49.686,160.124
C00744=1022.355,402.457,-153.988,173.325,49.685,160.121
C00745=1022.345,402.211,-153.943,173.313,49.683,160.119
C00746=1022.335,401.965,-153.898,173.301,49.682,160.117
C00747=1022.325,401.720,-153.853,173.290,49.681,160.115
C00748=1022.315,401.474,-153.808,173.278,49.680,160.113
C00749=1022.305,401.227,-153.764,173.268,49.679,160.110
C00750=1022.295,400.982,-153.719,173.256,49.678,160.108
C00751=1022.285,400.737,-153.675,173.244,49.677,160.106
C00752=1022.275,400.491,-153.630,173.233,49.676,160.104
C00753=1022.265,400.245,-153.586,173.222,49.674,160.102
C00754=1022.255,399.999,-153.541,173.210,49.673,160.100
C00755=1022.245,399.754,-153.496,173.199,49.673,160.098
C00756=1022.235,399.508,-153.453,173.189,49.671,160.096
C00757=1022.225,399.262,-153.408,173.177,49.670,160.093
C00758=1022.216,399.016,-153.364,173.165,49.669,160.091
C00759=1022.205,398.771,-153.320,173.155,49.668,160.089
C00760=1022.196,398.525,-153.276,173.144,49.667,160.087
C00761=1022.187,398.279,-153.231,173.133,49.666,160.085
C00762=1022.176,398.033,-153.187,173.122,49.665,160.083
C00763=1022.167,397.787,-153.143,173.111,49.664,160.081
C00764=1022.157,397.541,-153.100,173.100,49.663,160.079
C00765=1022.147,397.295,-153.055,173.088,49.662,160.077
C00766=1022.137,397.050,-153.012,173.078,49.661,160.075
C00767=1022.124,396.743,-152.957,173.064,49.660,160.073
C00768=1022.112,396.437,-152.903,173.051,49.659,160.070
C00769=1022.101,396.131,-152.848,173.037,49.658,160.068
C00770=1022.088,395.823,-152.793,173.024,49.657,160.065
C00771=1022.079,395.578,-152.750,173.013,49.657,160.063
C00772=1022.069,395.332,-152.706,173.003,49.655,160.061
C00773=1022.059,395.086,-152.663,172.991,49.655,160.059
C00774=1022.049,394.840,-152.620,172.981,49.654,160.057
C00775=1022.040,394.594,-152.576,172.970,49.654,160.055
C00776=1022.030,394.349,-152.533,172.960,49.653,160.054
C00777=1022.021,394.103,-152.489,172.949,49.652,160.052
C00778=1022.011,393.856,-152.446,172.938,49.651,160.050
C00779=1022.002,393.611,-152.402,172.928,49.650,160.048
C00780=1021.992,393.364,-152.359,172.918,49.650,160.046
C00781=1021.982,393.118,-152.316,172.906,49.649,160.044
C00782=1021.973,392.873,-152.272,172.896,49.648,160.042
C00783=1021.964,392.627,-152.229,172.886,49.648,160.040
C00784=1021.954,392.380,-152.186,172.876,49.647,160.039
C00785=1021.945,392.135,-152.143,172.865,49.647,160.037
C00786=1021.935,391.888,-152.100,172.855,49.646,160.035
C00787=1021.926,391.642,-152.057,172.845,49.645,160.033
C00788=1021.916,391.396,-152.015,172.834,49.645,160.031
C00789=1021.907,391.149,-151.971,172.824,49.645,160.029
C00790=1021.897,390.904,-151.928,172.813,49.644,160.028
C00791=1021.888,390.658,-151.886,172.803,49.643,160.026
C00792=1021.878,390.412,-151.843,172.793,49.643,160.024
C00793=1021.870,390.166,-151.800,172.783,49.642,160.022
C00794=1021.860,389.919,-151.757,172.772,49.642,160.020
C00795=1021.851,389.674,-151.715,172.762,49.641,160.019
C00796=1021.841,389.427,-151.672,172.752,49.641,160.017
C00797=1021.832,389.181,-151.629,172.742,49.640,160.015
C00798=1021.823,388.935,-151.586,172.732,49.640,160.014
C00799=1021.813,388.689,-151.543,172.722,49.639,160.012
C00800=1021.804,388.443,-151.502,172.712,49.639,160.010
C00801=1021.795,388.197,-151.459,172.702,49.639,160.008
C00802=1021.786,387.950,-151.416,172.692,49.639,160.007
C00803=1021.777,387.704,-151.374,172.681,49.638,160.005
C00804=1021.768,387.458,-151.332,172.671,49.637,160.003
C00805=1021.759,387.212,-151.289,172.662,49.637,160.001
C00806=1021.749,386.965,-151.247,172.652,49.637,160.000
C00807=1021.740,386.720,-151.205,172.642,49.636,159.998
C00808=1021.731,386.473,-151.163,172.632,49.636,159.996
C00809=1021.722,386.227,-151.121,172.622,49.636,159.995
C00810=1021.713,385.981,-151.079,172.612,49.636,159.993
C00811=1021.703,385.735,-151.037,172.602,49.635,159.991
C00812=1021.694,385.488,-150.994,172.593,49.635,159.990
C00813=1021.685,385.242,-150.953,172.583,49.635,159.988
C00814=1021.676,384.995,-150.911,172.573,49.635,159.987
C00815=1021.667,384.750,-150.869,172.563,49.635,159.985
C00816=1021.658,384.503,-150.827,172.554,49.634,159.983
C00817=1021.649,384.257,-150.785,172.545,49.634,159.982
C00818=1021.639,384.011,-150.744,172.535,49.634,159.980
C00819=1021.630,383.765,-150.702,172.526,49.634,159.979
C00820=1021.621,383.518,-150.661,172.516,49.634,159.977
C00821=1021.612,383.272,-150.619,172.506,49.634,159.975
C00822=1021.604,383.026,-150.577,172.496,49.634,159.974
C00823=1021.595,382.779,-150.535,172.487,49.634,159.972
C00824=1021.585,382.533,-150.494,172.477,49.634,159.971
C00825=1021.576,382.287,-150.453,172.468,49.633,159.969
C00826=1021.567,382.040,-150.411,172.459,49.634,159.968
C00827=1021.558,381.771,-150.366,172.448,49.634,159.966
C00828=1021.548,381.501,-150.321,172.438,49.633,159.964
C00829=1021.538,381.233,-150.276,172.427,49.634,159.963
C00830=1021.529,380.963,-150.230,172.418,49.634,159.961
C00831=1021.520,380.717,-150.189,172.408,49.634,159.960
C00832=1021.511,380.470,-150.147,172.398,49.633,159.958
C00833=1021.502,380.223,-150.106,172.389,49.634,159.957
C00834=1021.493,379.978,-150.065,172.380,49.634,159.955
C00835=1021.484,379.731,-150.024,172.371,49.634,159.954
C00836=1021.475,379.485,-149.983,172.361,49.634,159.952
C00837=1021.467,379.238,-149.942,172.352,49.634,159.951
C00838=1021.458,378.992,-149.900,172.343,49.634,159.949
C00839=1021.449,378.745,-149.860,172.333,49.634,159.948
C00840=1021.441,378.500,-149.818,172.324,49.634,159.946
C00841=1021.432,378.253,-149.777,172.315,49.634,159.945
C00842=1021.423,378.006,-149.736,172.306,49.635,159.943
C00843=1021.415,377.760,-149.695,172.297,49.634,159.942
C00844=1021.407,377.513,-149.654,172.288,49.635,159.941
C00845=1021.398,377.267,-149.614,172.278,49.635,159.939
C00846=1021.389,377.021,-149.572,172.270,49.635,159.938
C00847=1021.381,376.774,-149.532,172.260,49.635,159.936
C00848=1021.372,376.527,-149.491,172.252,49.635,159.935
C00849=1021.364,376.281,-149.450,172.243,49.636,159.934
C00850=1021.355,376.035,-149.410,172.233,49.636,159.932
C00851=1021.346,375.788,-149.369,172.225,49.636,159.931
C00852=1021.337,375.542,-149.329,172.216,49.637,159.930
C00853=1021.329,375.295,-149.288,172.207,49.637,159.928
C00854=1021.320,375.049,-149.248,172.198,49.637,159.927
C00855=1021.312,374.801,-149.207,172.189,49.638,159.925
C00856=1021.303,374.555,-149.167,172.180,49.638,159.924
C00857=1021.295,374.309,-149.127,172.171,49.639,159.923
C00858=1021.286,374.062,-149.086,172.162,49.639,159.921
C00859=1021.277,373.816,-149.046,172.153,49.640,159.920
C00860=1021.268,373.568,-149.006,172.145,49.640,159.919
C00861=1021.260,373.322,-148.965,172.136,49.640,159.918
C00862=1021.252,373.076,-148.925,172.127,49.640,159.916
C00863=1021.243,372.829,-148.885,172.118,49.641,159.915
C00864=1021.235,372.583,-148.845,172.110,49.641,159.914
C00865=1021.227,372.336,-148.805,172.101,49.642,159.912
C00866=1021.218,372.090,-148.765,172.092,49.643,159.911
C00867=1021.210,371.842,-148.725,172.083,49.643,159.910
C00868=1021.201,371.596,-148.685,172.075,49.643,159.908
C00869=1021.193,371.349,-148.645,172.067,49.644,159.907
C00870=1021.184,371.103,-148.605,172.058,49.645,159.906
C00871=1021.176,370.856,-148.564,172.049,49.645,159.905
C00872=1021.168,370.609,-148.525,172.040,49.645,159.903
C00873=1021.159,370.363,-148.485,172.032,49.646,159.902
C00874=1021.151,370.116,-148.445,172.023,49.647,159.901
C00875=1021.143,369.870,-148.406,172.015,49.647,159.900
C00876=1021.135,369.623,-148.365,172.006,49.648,159.899
C00877=1021.126,369.377,-148.326,171.997,49.649,159.897
C00878=1021.119,369.130,-148.286,171.989,49.649,159.896
C00879=1021.110,368.883,-148.246,171.981,49.650,159.895
C00880=1021.102,368.636,-148.206,171.972,49.651,159.894
C00881=1021.093,368.389,-148.167,171.964,49.651,159.893
C00882=1021.085,368.143,-148.126,171.956,49.652,159.891
C00883=1021.077,367.896,-148.087,171.947,49.652,159.890
C00884=1021.069,367.649,-148.048,171.938,49.653,159.889
C00885=1021.060,367.402,-148.009,171.930,49.653,159.888
C00886=1021.053,367.155,-147.969,171.921,49.654,159.887
C00887=1021.044,366.909,-147.930,171.913,49.655,159.886
C00888=1021.036,366.662,-147.891,171.905,49.656,159.884
C00889=1021.028,366.414,-147.851,171.896,49.657,159.883
C00890=1021.019,366.167,-147.812,171.888,49.658,159.882
C00891=1021.011,365.920,-147.773,171.880,49.658,159.881
C00892=1021.003,365.674,-147.734,171.872,49.659,159.880
C00893=1020.994,365.427,-147.694,171.863,49.660,159.879
C00894=1020.986,365.180,-147.656,171.855,49.661,159.878
C00895=1020.979,364.934,-147.616,171.847,49.662,159.877
C00896=1020.971,364.686,-147.578,171.839,49.663,159.875
C00897=1020.962,364.440,-147.538,171.830,49.663,159.874
C00898=1020.954,364.193,-147.500,171.822,49.664,159.873
C00899=1020.946,363.946,-147.460,171.814,49.665,159.872
C00900=1020.937,363.699,-147.422,171.807,49.666,159.871
C00901=1020.930,363.453,-147.383,171.798,49.668,159.870
C00902=1020.922,363.205,-147.343,171.790,49.668,159.869
C00903=1020.914,362.959,-147.304,171.782,49.669,159.868
C00904=1020.906,362.712,-147.266,171.774,49.670,159.867
C00905=1020.898,362.465,-147.227,171.766,49.671,159.866
C00906=1020.890,362.218,-147.188,171.758,49.672,159.865
C00907=1020.881,361.971,-147.149,171.749,49.673,159.863
C00908=1020.874,361.725,-147.111,171.741,49.674,159.862
C00909=1020.866,361.478,-147.071,171.734,49.675,159.861
C00910=1020.858,361.231,-147.033,171.726,49.676,159.861
C00911=1020.850,360.984,-146.994,171.718,49.677,159.859
C00912=1020.842,360.737,-146.956,171.710,49.678,159.858
C00913=1020.835,360.490,-146.918,171.702,49.679,159.857
C00914=1020.826,360.244,-146.878,171.695,49.680,159.856
C00915=1020.818,359.997,-146.840,171.686,49.681,159.855
C00916=1020.811,359.750,-146.801,171.678,49.683,159.854
C00917=1020.802,359.503,-146.763,171.670,49.684,159.853
C00918=1020.795,359.256,-146.724,171.662,49.685,159.852
C00919=1020.787,359.008,-146.687,171.655,49.686,159.851
C00920=1020.779,358.762,-146.648,171.647,49.687,159.850
C00921=1020.771,358.515,-146.610,171.639,49.688,159.850
C00922=1020.764,358.268,-146.572,171.631,49.689,159.849
C00923=1020.756,358.021,-146.533,171.624,49.690,159.848
C00924=1020.748,357.774,-146.495,171.616,49.691,159.847
C00925=1020.739,357.527,-146.457,171.608,49.693,159.846
C00926=1020.732,357.280,-146.419,171.600,49.694,159.845
C00927=1020.724,357.033,-146.381,171.592,49.695,159.844
C00928=1020.717,356.786,-146.343,171.584,49.697,159.843
C00929=1020.708,356.539,-146.304,171.576,49.698,159.842
C00930=1020.701,356.292,-146.266,171.569,49.699,159.841
C00931=1020.693,356.046,-146.229,171.561,49.700,159.840
C00932=1020.685,355.798,-146.191,171.554,49.702,159.839
C00933=1020.677,355.551,-146.153,171.546,49.703,159.838
C00934=1020.669,355.304,-146.114,171.538,49.704,159.837
C00935=1020.662,355.057,-146.077,171.531,49.706,159.836
C00936=1020.654,354.811,-146.039,171.523,49.707,159.835
C00937=1020.647,354.563,-146.002,171.516,49.709,159.835
C00938=1020.638,354.316,-145.963,171.508,49.710,159.834
C00939=1020.631,354.069,-145.926,171.500,49.711,159.833
C00940=1020.623,353.822,-145.889,171.493,49.713,159.832
C00941=1020.615,353.574,-145.851,171.485,49.714,159.831
C00942=1020.608,353.328,-145.813,171.477,49.715,159.830
C00943=1020.600,353.085,-145.776,171.471,49.717,159.829
C00944=1020.592,352.841,-145.739,171.463,49.718,159.829
C00945=1020.585,352.598,-145.702,171.456,49.720,159.828
C00946=1020.578,352.354,-145.665,171.448,49.721,159.827
C00947=1020.570,352.111,-145.628,171.441,49.722,159.826
C00948=1020.562,351.868,-145.591,171.433,49.724,159.825
C00949=1020.555,351.624,-145.555,171.426,49.726,159.824
C00950=1020.546,351.381,-145.518,171.419,49.727,159.824
C00951=1020.539,351.133,-145.480,171.412,49.728,159.823
C00952=1020.532,350.886,-145.442,171.404,49.730,159.822
C00953=1020.524,350.639,-145.406,171.397,49.732,159.821
C00954=1020.517,350.392,-145.368,171.389,49.733,159.820
C00955=1020.509,350.145,-145.330,171.382,49.735,159.819
C00956=1020.502,349.898,-145.294,171.375,49.736,159.819
C00957=1020.495,349.651,-145.257,171.367,49.738,159.818
C00958=1020.487,349.404,-145.220,171.360,49.740,159.817
C00959=1020.479,349.157,-145.182,171.353,49.741,159.816
C00960=1020.472,348.910,-145.145,171.346,49.742,159.815
C00961=1020.464,348.663,-145.108,171.338,49.744,159.815
C00962=1020.457,348.415,-145.071,171.331,49.746,159.814
C00963=1020.449,348.168,-145.034,171.323,49.748,159.813
C00964=1020.442,347.921,-144.997,171.316,49.749,159.812
C00965=1020.434,347.674,-144.960,171.309,49.751,159.812
C00966=1020.427,347.426,-144.923,171.302,49.752,159.811
C00967=1020.419,347.180,-144.886,171.295,49.754,159.810
C00968=1020.412,346.932,-144.849,171.287,49.756,159.809
C00969=1020.404,346.685,-144.812,171.280,49.758,159.809
C00970=1020.396,346.438,-144.776,171.273,49.760,159.808
C00971=1020.389,346.190,-144.738,171.266,49.762,159.807
C00972=1020.381,345.943,-144.702,171.258,49.763,159.806
C00973=1020.373,345.696,-144.665,171.252,49.765,159.806
C00974=1020.367,345.448,-144.628,171.245,49.767,159.805
C00975=1020.359,345.202,-144.592,171.237,49.769,159.804
C00976=1020.352,344.955,-144.556,171.230,49.771,159.804
C00977=1020.345,344.707,-144.519,171.223,49.772,159.803
C00978=1020.337,344.460,-144.482,171.217,49.774,159.802
C00979=1020.330,344.212,-144.445,171.209,49.776,159.802
C00980=1020.323,343.966,-144.409,171.202,49.778,159.801
C00981=1020.315,343.719,-144.372,171.195,49.780,159.800
C00982=1020.308,343.471,-144.335,171.187,49.782,159.799
C00983=1020.300,343.224,-144.299,171.181,49.783,159.799
C00984=1020.293,342.977,-144.263,171.174,49.786,159.798
C00985=1020.285,342.730,-144.227,171.167,49.787,159.797
C00986=1020.278,342.482,-144.190,171.160,49.790,159.797
C00987=1020.270,342.235,-144.153,171.153,49.791,159.796
C00988=1020.263,341.988,-144.118,171.146,49.793,159.796
C00989=1020.256,341.740,-144.081,171.139,49.795,159.795
C00990=1020.249,341.493,-144.045,171.132,49.797,159.794
C00991=1020.242,341.246,-144.009,171.125,49.799,159.793
C00992=1020.234,340.999,-143.973,171.118,49.801,159.793
C00993=1020.227,340.751,-143.936,171.111,49.804,159.792
C00994=1020.220,340.504,-143.900,171.104,49.805,159.792
C00995=1020.212,340.257,-143.864,171.098,49.807,159.791
C00996=1020.205,340.009,-143.828,171.091,49.809,159.790
C00997=1020.198,339.762,-143.792,171.084,49.811,159.790
C00998=1020.191,339.515,-143.756,171.076,49.814,159.789
C00999=1020.184,339.268,-143.720,171.070,49.815,159.788
C01000=1020.176,339.020,-143.683,171.063,49.817,159.788
C01001=1020.169,338.773,-143.648,171.056,49.820,159.787
C01002=1020.162,338.525,-143.612,171.050,49.822,159.787
C01003=1020.155,338.281,-143.577,171.043,49.824,159.786
C01004=1020.147,338.036,-143.541,171.036,49.826,159.786
C01005=1020.140,337.791,-143.506,171.030,49.828,159.785
C01006=1020.133,337.546,-143.470,171.023,49.830,159.784
C01007=1020.125,337.301,-143.435,171.016,49.833,159.784
C01008=1020.118,337.056,-143.400,171.010,49.835,159.783
C01009=1020.112,336.811,-143.364,171.002,49.837,159.783
C01010=1020.104,336.566,-143.328,170.995,49.839,159.782
C01011=1020.097,336.318,-143.293,170.989,49.841,159.782
C01012=1020.090,336.071,-143.257,170.982,49.844,159.781
C01013=1020.083,335.824,-143.222,170.975,49.846,159.780
C01014=1020.076,335.576,-143.187,170.969,49.848,159.780
C01015=1020.069,335.329,-143.151,170.962,49.850,159.779
C01016=1020.062,335.081,-143.115,170.955,49.853,159.779
C01017=1020.054,334.834,-143.079,170.949,49.855,159.778
C01018=1020.047,334.587,-143.044,170.942,49.857,159.778
C01019=1020.041,334.339,-143.009,170.935,49.859,159.777
C01020=1020.033,334.092,-142.973,170.930,49.862,159.777
C01021=1020.026,333.844,-142.938,170.923,49.864,159.776
C01022=1020.019,333.597,-142.902,170.916,49.867,159.776
C01023=1020.012,333.350,-142.867,170.910,49.869,159.775
C01024=1020.005,333.102,-142.831,170.903,49.871,159.775
C01025=1019.997,332.855,-142.797,170.896,49.873,159.774
C01026=1019.991,332.608,-142.761,170.890,49.876,159.774
C01027=1019.983,332.360,-142.726,170.883,49.879,159.773
C01028=1019.977,332.112,-142.691,170.877,49.881,159.773
C01029=1019.969,331.865,-142.656,170.870,49.884,159.772
C01030=1019.962,331.618,-142.621,170.863,49.886,159.772
C01031=1019.955,331.370,-142.586,170.857,49.889,159.771
C01032=1019.948,331.123,-142.551,170.850,49.891,159.771
C01033=1019.941,330.876,-142.516,170.843,49.893,159.770
C01034=1019.934,330.628,-142.481,170.838,49.896,159.770
C01035=1019.927,330.381,-142.446,170.831,49.898,159.769
C01036=1019.920,330.133,-142.411,170.825,49.901,159.769
C01037=1019.912,329.886,-142.376,170.818,49.903,159.768
C01038=1019.905,329.638,-142.341,170.811,49.906,159.768
C01039=1019.899,329.391,-142.305,170.805,49.908,159.768
C01040=1019.891,329.143,-142.272,170.799,49.911,159.767
C01041=1019.885,328.896,-142.236,170.792,49.914,159.767
C01042=1019.878,328.649,-142.201,170.786,49.916,159.766
C01043=1019.871,328.401,-142.166,170.779,49.919,159.766
C01044=1019.864,328.154,-142.132,170.773,49.921,159.765
C01045=1019.857,327.906,-142.097,170.767,49.924,159.765
C01046=1019.850,327.659,-142.062,170.761,49.926,159.765
C01047=1019.843,327.412,-142.028,170.754,49.929,159.764
C01048=1019.836,327.164,-141.993,170.747,49.932,159.764
C01049=1019.830,326.916,-141.958,170.741,49.934,159.763
C01050=1019.823,326.669,-141.923,170.735,49.937,159.763
C01051=1019.816,326.421,-141.889,170.729,49.940,159.763
C01052=1019.808,326.174,-141.854,170.722,49.942,159.762
C01053=1019.802,325.926,-141.820,170.715,49.945,159.762
C01054=1019.795,325.679,-141.786,170.710,49.948,159.761
C01055=1019.787,325.432,-141.752,170.703,49.951,159.761
C01056=1019.780,325.184,-141.718,170.697,49.954,159.761
C01057=1019.773,324.936,-141.683,170.691,49.957,159.760
C01058=1019.766,324.689,-141.649,170.684,49.960,159.760
C01059=1019.759,324.441,-141.615,170.678,49.962,159.760
C01060=1019.752,324.193,-141.581,170.672,49.965,159.759
C01061=1019.745,323.946,-141.546,170.665,49.968,159.759
C01062=1019.738,323.699,-141.512,170.660,49.971,159.759
C01063=1019.730,323.451,-141.478,170.653,49.974,159.758
C01064=1019.723,323.205,-141.444,170.647,49.977,159.758
C01065=1019.717,322.957,-141.410,170.641,49.980,159.757
C01066=1019.710,322.709,-141.376,170.635,49.982,159.757
C01067=1019.703,322.463,-141.342,170.628,49.985,159.757
C01068=1019.696,322.215,-141.308,170.622,49.988,159.756
C01069=1019.689,321.968,-141.275,170.616,49.991,159.756
C01070=1019.682,321.720,-141.241,170.610,49.995,159.756
C01071=1019.674,321.473,-141.206,170.604,49.997,159.756
C01072=1019.668,321.226,-141.172,170.597,50.000,159.755
C01073=1019.661,320.978,-141.138,170.592,50.003,159.755
C01074=1019.654,320.731,-141.105,170.585,50.006,159.755
C01075=1019.648,320.483,-141.070,170.579,50.009,159.754
C01076=1019.641,320.236,-141.037,170.573,50.012,159.754
C01077=1019.634,319.988,-141.003,170.567,50.015,159.754
C01078=1019.627,319.740,-140.969,170.561,50.018,159.753
C01079=1019.620,319.492,-140.935,170.554,50.021,159.753
C01080=1019.614,319.245,-140.902,170.549,50.024,159.753
C01081=1019.607,318.997,-140.868,170.542,50.027,159.752
C01082=1019.599,318.749,-140.834,170.537,50.030,159.752
C01083=1019.594,318.502,-140.800,170.530,50.034,159.752
C01084=1019.586,318.254,-140.766,170.525,50.036,159.752
C01085=1019.579,318.007,-140.732,170.518,50.039,159.751
C01086=1019.573,317.760,-140.699,170.513,50.043,159.751
C01087=1019.566,317.511,-140.665,170.506,50.046,159.751
C01088=1019.560,317.264,-140.632,170.500,50.048,159.750
C01089=1019.553,317.016,-140.598,170.494,50.052,159.750
C01090=1019.545,316.769,-140.564,170.489,50.055,159.750
C01091=1019.540,316.521,-140.531,170.482,50.058,159.750
C01092=1019.533,316.273,-140.497,170.477,50.061,159.750
C01093=1019.526,316.026,-140.464,170.470,50.065,159.749
C01094=1019.519,315.778,-140.430,170.465,50.067,159.749
C01095=1019.513,315.531,-140.396,170.458,50.071,159.749
C01096=1019.506,315.283,-140.363,170.453,50.074,159.749
C01097=1019.500,315.035,-140.330,170.447,50.077,159.748
C01098=1019.493,314.788,-140.296,170.441,50.080,159.748
C01099=1019.486,314.540,-140.263,170.435,50.084,159.748
C01100=1019.480,314.292,-140.229,170.429,50.086,159.748
C01101=1019.473,314.045,-140.195,170.423,50.090,159.747
C01102=1019.466,313.797,-140.162,170.417,50.093,159.747
C01103=1019.460,313.550,-140.129,170.411,50.096,159.747
C01104=1019.454,313.301,-140.095,170.405,50.100,159.747
C01105=1019.447,313.054,-140.062,170.400,50.102,159.746
C01106=1019.441,312.807,-140.029,170.394,50.106,159.746
C01107=1019.434,312.559,-139.995,170.388,50.109,159.746
C01108=1019.428,312.311,-139.962,170.382,50.112,159.746
C01109=1019.421,312.064,-139.928,170.376,50.116,159.746
C01110=1019.415,311.816,-139.895,170.370,50.119,159.745
C01111=1019.408,311.568,-139.862,170.365,50.122,159.745
C01112=1019.402,311.321,-139.829,170.358,50.126,159.745
C01113=1019.395,311.073,-139.795,170.353,50.129,159.745
C01114=1019.389,310.825,-139.763,170.348,50.132,159.745
C01115=1019.383,310.578,-139.729,170.341,50.136,159.745
C01116=1019.376,310.330,-139.696,170.336,50.138,159.744
C01117=1019.370,310.082,-139.663,170.329,50.142,159.744
C01118=1019.364,309.835,-139.629,170.324,50.145,159.744
C01119=1019.356,309.588,-139.597,170.318,50.149,159.744
C01120=1019.350,309.339,-139.564,170.313,50.152,159.744
C01121=1019.343,309.092,-139.532,170.306,50.156,159.743
C01122=1019.337,308.844,-139.500,170.301,50.159,159.743
C01123=1019.329,308.600,-139.468,170.295,50.163,159.743
C01124=1019.323,308.355,-139.435,170.289,50.166,159.743
C01125=1019.316,308.110,-139.403,170.284,50.171,159.743
C01126=1019.310,307.865,-139.370,170.278,50.174,159.743
C01127=1019.303,307.621,-139.339,170.273,50.177,159.743
C01128=1019.296,307.376,-139.306,170.267,50.181,159.743
C01129=1019.290,307.132,-139.275,170.261,50.184,159.743
C01130=1019.283,306.888,-139.243,170.255,50.188,159.742
C01131=1019.277,306.639,-139.210,170.250,50.192,159.742
C01132=1019.270,306.391,-139.177,170.244,50.196,159.742
C01133=1019.263,306.144,-139.145,170.239,50.199,159.742
C01134=1019.257,305.896,-139.112,170.233,50.203,159.742
C01135=1019.250,305.648,-139.081,170.228,50.207,159.742
C01136=1019.244,305.401,-139.048,170.221,50.210,159.742
C01137=1019.237,305.153,-139.016,170.216,50.214,159.742
C01138=1019.230,304.905,-138.983,170.210,50.217,159.741
C01139=1019.224,304.657,-138.951,170.205,50.221,159.742
C01140=1019.217,304.410,-138.919,170.199,50.225,159.741
C01141=1019.211,304.161,-138.887,170.193,50.228,159.741
C01142=1019.204,303.914,-138.855,170.187,50.233,159.741
C01143=1019.197,303.666,-138.822,170.182,50.236,159.741
C01144=1019.191,303.418,-138.790,170.176,50.240,159.741
C01145=1019.184,303.171,-138.758,170.171,50.244,159.741
C01146=1019.178,302.923,-138.726,170.165,50.247,159.741
C01147=1019.171,302.675,-138.693,170.160,50.251,159.741
C01148=1019.165,302.427,-138.661,170.154,50.255,159.741
C01149=1019.158,302.179,-138.629,170.149,50.259,159.741
C01150=1019.152,301.931,-138.597,170.142,50.263,159.741
C01151=1019.145,301.683,-138.564,170.138,50.267,159.741
C01152=1019.139,301.436,-138.533,170.132,50.270,159.741
C01153=1019.132,301.188,-138.500,170.126,50.274,159.741
C01154=1019.126,300.940,-138.469,170.121,50.278,159.741
C01155=1019.119,300.692,-138.436,170.115,50.282,159.741
C01156=1019.113,300.445,-138.405,170.110,50.285,159.740
C01157=1019.107,300.196,-138.372,170.104,50.290,159.740
C01158=1019.100,299.949,-138.340,170.099,50.293,159.740
C01159=1019.094,299.701,-138.308,170.093,50.297,159.740
C01160=1019.088,299.453,-138.277,170.088,50.301,159.740
C01161=1019.081,299.206,-138.244,170.083,50.305,159.740
C01162=1019.075,298.958,-138.212,170.077,50.309,159.740
C01163=1019.068,298.710,-138.181,170.072,50.313,159.740
C01164=1019.062,298.462,-138.148,170.066,50.317,159.740
C01165=1019.056,298.214,-138.116,170.061,50.321,159.740
C01166=1019.049,297.966,-138.085,170.055,50.325,159.740
C01167=1019.044,297.718,-138.053,170.050,50.328,159.740
C01168=1019.037,297.470,-138.021,170.044,50.333,159.740
C01169=1019.031,297.223,-137.989,170.039,50.337,159.740
C01170=1019.024,296.975,-137.958,170.034,50.340,159.740
C01171=1019.018,296.727,-137.926,170.028,50.344,159.740
C01172=1019.012,296.479,-137.894,170.023,50.348,159.740
C01173=1019.006,296.231,-137.862,170.017,50.353,159.740
C01174=1019.000,295.984,-137.830,170.012,50.356,159.740
C01175=1018.994,295.736,-137.799,170.007,50.360,159.740
C01176=1018.987,295.488,-137.766,170.001,50.364,159.740
C01177=1018.981,295.240,-137.735,169.996,50.368,159.740
C01178=1018.975,294.992,-137.703,169.990,50.373,159.740
C01179=1018.968,294.745,-137.672,169.985,50.377,159.740
C01180=1018.962,294.496,-137.640,169.979,50.380,159.740
C01181=1018.956,294.249,-137.608,169.974,50.384,159.740
C01182=1018.950,294.000,-137.576,169.969,50.388,159.740
C01183=1018.944,293.765,-137.547,169.964,50.392,159.740
C01184=1018.939,293.529,-137.517,169.960,50.396,159.740
C01185=1018.932,293.293,-137.486,169.954,50.401,159.740
C01186=1018.927,293.057,-137.456,169.948,50.404,159.740
C01187=1018.921,292.821,-137.427,169.943,50.408,159.740
C01188=1018.915,292.585,-137.397,169.939,50.412,159.740
C01189=1018.908,292.350,-137.367,169.934,50.416,159.741
C01190=1018.903,292.114,-137.337,169.929,50.420,159.741
C01191=1018.896,291.866,-137.307,169.923,50.425,159.741
C01192=1018.890,291.618,-137.275,169.918,50.429,159.741
C01193=1018.884,291.371,-137.243,169.913,50.434,159.741
C01194=1018.878,291.123,-137.212,169.908,50.438,159.741
C01195=1018.871,290.874,-137.181,169.902,50.442,159.741
C01196=1018.865,290.627,-137.150,169.897,50.446,159.741
C01197=1018.859,290.378,-137.119,169.891,50.450,159.741
C01198=1018.852,290.130,-137.088,169.887,50.455,159.741
C01199=1018.846,289.883,-137.058,169.881,50.459,159.741
C01200=1018.839,289.635,-137.026,169.876,50.463,159.741
C01201=1018.833,289.386,-136.996,169.871,50.467,159.742
C01202=1018.827,289.139,-136.964,169.865,50.472,159.742
C01203=1018.820,288.890,-136.934,169.861,50.476,159.742
C01204=1018.814,288.642,-136.902,169.855,50.481,159.742
C01205=1018.809,288.394,-136.871,169.850,50.485,159.742
C01206=1018.802,288.147,-136.840,169.844,50.490,159.742
C01207=1018.796,287.899,-136.810,169.839,50.494,159.742
C01208=1018.789,287.651,-136.778,169.834,50.499,159.742
C01209=1018.784,287.403,-136.748,169.829,50.503,159.742
C01210=1018.777,287.154,-136.717,169.824,50.508,159.743
C01211=1018.771,286.907,-136.686,169.819,50.512,159.743
C01212=1018.765,286.659,-136.655,169.813,50.517,159.743
C01213=1018.758,286.410,-136.625,169.808,50.521,159.743
C01214=1018.752,286.163,-136.594,169.803,50.526,159.743
C01215=1018.746,285.914,-136.563,169.798,50.530,159.743
C01216=1018.740,285.667,-136.532,169.792,50.535,159.743
C01217=1018.733,285.418,-136.502,169.788,50.539,159.744
C01218=1018.727,285.171,-136.471,169.783,50.544,159.744
C01219=1018.721,284.922,-136.440,169.777,50.548,159.744
C01220=1018.715,284.675,-136.410,169.773,50.553,159.744
C01221=1018.708,284.427,-136.380,169.767,50.557,159.744
C01222=1018.702,284.179,-136.349,169.762,50.562,159.744
C01223=1018.696,283.931,-136.319,169.757,50.567,159.745
C01224=1018.690,283.682,-136.288,169.752,50.571,159.745
C01225=1018.683,283.435,-136.258,169.747,50.576,159.745
C01226=1018.677,283.186,-136.228,169.741,50.581,159.745
C01227=1018.671,282.938,-136.197,169.736,50.585,159.745
C01228=1018.665,282.690,-136.167,169.731,50.590,159.745
C01229=1018.659,282.442,-136.136,169.726,50.595,159.746
C01230=1018.652,282.195,-136.106,169.721,50.600,159.746
C01231=1018.646,281.946,-136.076,169.716,50.604,159.746
C01232=1018.640,281.698,-136.045,169.710,50.609,159.746
C01233=1018.634,281.450,-136.015,169.706,50.614,159.746
C01234=1018.627,281.202,-135.985,169.700,50.619,159.747
C01235=1018.621,280.954,-135.955,169.696,50.623,159.747
C01236=1018.615,280.706,-135.924,169.690,50.628,159.747
C01237=1018.609,280.458,-135.893,169.686,50.632,159.747
C01238=1018.602,280.210,-135.864,169.680,50.637,159.747
C01239=1018.596,279.961,-135.834,169.676,50.642,159.748
C01240=1018.591,279.713,-135.803,169.670,50.647,159.748
C01241=1018.585,279.466,-135.773,169.666,50.652,159.748
C01242=1018.578,279.217,-135.743,169.660,50.657,159.748
C01243=1018.572,278.987,-135.715,169.655,50.661,159.748
C01244=1018.566,278.758,-135.687,169.651,50.666,159.749
C01245=1018.561,278.529,-135.659,169.646,50.670,159.749
C01246=1018.555,278.299,-135.632,169.641,50.674,159.749
C01247=1018.550,278.069,-135.603,169.637,50.679,159.749
C01248=1018.544,277.839,-135.576,169.632,50.684,159.750
C01249=1018.539,277.610,-135.548,169.628,50.688,159.750
C01250=1018.533,277.380,-135.520,169.623,50.693,159.750
C01251=1018.527,277.132,-135.490,169.619,50.697,159.750
C01252=1018.520,276.884,-135.460,169.613,50.702,159.750
C01253=1018.515,276.636,-135.430,169.609,50.707,159.751
C01254=1018.509,276.388,-135.400,169.603,50.712,159.751
C01255=1018.503,276.140,-135.371,169.599,50.717,159.751
C01256=1018.496,275.891,-135.340,169.593,50.722,159.751
C01257=1018.490,275.643,-135.311,169.589,50.727,159.752
C01258=1018.484,275.395,-135.281,169.584,50.732,159.752
C01259=1018.478,275.147,-135.251,169.579,50.737,159.752
C01260=1018.472,274.899,-135.221,169.574,50.742,159.752
C01261=1018.465,274.650,-135.192,169.569,50.747,159.753
C01262=1018.460,274.402,-135.161,169.564,50.752,159.753
C01263=1018.453,274.154,-135.132,169.560,50.757,159.753
C01264=1018.448,273.906,-135.103,169.554,50.762,159.754
C01265=1018.441,273.658,-135.073,169.549,50.767,159.754
C01266=1018.436,273.410,-135.043,169.545,50.773,159.754
C01267=1018.429,273.162,-135.013,169.539,50.778,159.754
C01268=1018.423,272.913,-134.984,169.535,50.782,159.755
C01269=1018.417,272.665,-134.955,169.530,50.788,159.755
C01270=1018.411,272.417,-134.924,169.525,50.793,159.755
C01271=1018.405,272.169,-134.895,169.520,50.798,159.756
C01272=1018.399,271.921,-134.865,169.516,50.803,159.756
C01273=1018.393,271.673,-134.836,169.510,50.808,159.756
C01274=1018.386,271.425,-134.807,169.506,50.813,159.756
C01275=1018.381,271.177,-134.777,169.501,50.819,159.757
C01276=1018.375,270.929,-134.748,169.495,50.824,159.757
C01277=1018.369,270.680,-134.718,169.491,50.829,159.758
C01278=1018.363,270.432,-134.689,169.486,50.834,159.758
C01279=1018.356,270.184,-134.659,169.482,50.840,159.758
C01280=1018.350,269.935,-134.630,169.476,50.845,159.758
C01281=1018.344,269.687,-134.601,169.472,50.850,159.759
C01282=1018.338,269.439,-134.571,169.467,50.855,159.759
C01283=1018.332,269.191,-134.542,169.462,50.861,159.760
C01284=1018.326,268.942,-134.513,169.457,50.866,159.760
C01285=1018.320,268.694,-134.483,169.452,50.872,159.760
C01286=1018.314,268.446,-134.454,169.447,50.876,159.760
C01287=1018.308,268.198,-134.425,169.442,50.882,159.761
C01288=1018.302,267.950,-134.396,169.438,50.887,159.761
C01289=1018.295,267.702,-134.367,169.433,50.893,159.761
C01290=1018.290,267.453,-134.337,169.428,50.898,159.762
C01291=1018.284,267.205,-134.308,169.423,50.903,159.762
C01292=1018.277,266.957,-134.279,169.418,50.909,159.762
C01293=1018.272,266.709,-134.251,169.414,50.914,159.763
C01294=1018.266,266.461,-134.221,169.409,50.920,159.763
C01295=1018.260,266.213,-134.192,169.404,50.925,159.764
C01296=1018.254,265.965,-134.163,169.400,50.930,159.764
C01297=1018.248,265.716,-134.135,169.395,50.936,159.764
C01298=1018.242,265.468,-134.106,169.390,50.941,159.765
C01299=1018.236,265.219,-134.076,169.385,50.947,159.765
C01300=1018.230,264.971,-134.047,169.380,50.952,159.765
C01301=1018.224,264.723,-134.018,169.376,50.958,159.766
C01302=1018.218,264.474,-133.990,169.371,50.964,159.766
C01303=1018.212,264.247,-133.963,169.366,50.968,159.767
C01304=1018.207,264.020,-133.937,169.362,50.974,159.767
C01305=1018.201,263.793,-133.910,169.358,50.978,159.767
C01306=1018.196,263.565,-133.884,169.354,50.984,159.768
C01307=1018.190,263.338,-133.857,169.349,50.989,159.768
C01308=1018.185,263.110,-133.830,169.345,50.994,159.769
C01309=1018.179,262.883,-133.804,169.341,50.999,159.769
C01310=1018.173,262.655,-133.779,169.337,51.004,159.769
C01311=1018.167,262.408,-133.750,169.332,51.010,159.770
C01312=1018.162,262.159,-133.720,169.326,51.015,159.770
C01313=1018.156,261.910,-133.692,169.322,51.021,159.770
C01314=1018.150,261.662,-133.663,169.317,51.026,159.771
C01315=1018.144,261.413,-133.635,169.313,51.032,159.771
C01316=1018.138,261.166,-133.606,169.308,51.037,159.772
C01317=1018.132,260.918,-133.577,169.303,51.043,159.772
C01318=1018.126,260.669,-133.549,169.299,51.049,159.772
C01319=1018.120,260.421,-133.519,169.294,51.054,159.773
C01320=1018.114,260.172,-133.491,169.289,51.061,159.773
C01321=1018.108,259.925,-133.462,169.285,51.066,159.774
C01322=1018.102,259.676,-133.434,169.280,51.072,159.774
C01323=1018.095,259.428,-133.406,169.275,51.078,159.775
C01324=1018.089,259.180,-133.377,169.271,51.083,159.775
C01325=1018.084,258.931,-133.349,169.266,51.090,159.776
C01326=1018.077,258.683,-133.322,169.261,51.096,159.776
C01327=1018.071,258.434,-133.293,169.256,51.101,159.777
C01328=1018.065,258.186,-133.264,169.252,51.107,159.777
C01329=1018.058,257.938,-133.237,169.248,51.113,159.778
C01330=1018.053,257.690,-133.209,169.243,51.119,159.778
C01331=1018.047,257.441,-133.180,169.237,51.125,159.778
C01332=1018.040,257.192,-133.153,169.234,51.131,159.779
C01333=1018.034,256.944,-133.124,169.229,51.137,159.779
C01334=1018.029,256.696,-133.096,169.224,51.142,159.780
C01335=1018.022,256.448,-133.068,169.219,51.149,159.780
C01336=1018.016,256.199,-133.040,169.215,51.154,159.781
C01337=1018.010,255.951,-133.012,169.210,51.161,159.782
C01338=1018.004,255.703,-132.984,169.205,51.167,159.782
C01339=1017.998,255.454,-132.956,169.200,51.172,159.782
C01340=1017.992,255.206,-132.928,169.197,51.178,159.783
C01341=1017.986,254.958,-132.899,169.192,51.184,159.783
C01342=1017.980,254.709,-132.871,169.187,51.191,159.784
C01343=1017.974,254.461,-132.843,169.182,51.197,159.784
C01344=1017.968,254.213,-132.815,169.178,51.203,159.785
C01345=1017.962,253.964,-132.787,169.173,51.208,159.785
C01346=1017.956,253.716,-132.759,169.169,51.215,159.786
C01347=1017.950,253.467,-132.731,169.164,51.221,159.786
C01348=1017.944,253.219,-132.703,169.160,51.227,159.787
C01349=1017.938,252.971,-132.675,169.155,51.233,159.787
C01350=1017.932,252.722,-132.647,169.150,51.239,159.788
C01351=1017.926,252.474,-132.620,169.145,51.245,159.788
C01352=1017.920,252.226,-132.591,169.142,51.251,159.789
C01353=1017.915,251.978,-132.563,169.137,51.258,159.790
C01354=1017.908,251.729,-132.536,169.132,51.263,159.790
C01355=1017.902,251.480,-132.508,169.127,51.270,159.791
C01356=1017.897,251.232,-132.480,169.123,51.275,159.791
C01357=1017.890,250.983,-132.452,169.119,51.282,159.792
C01358=1017.885,250.735,-132.424,169.114,51.288,159.792
C01359=1017.878,250.487,-132.397,169.109,51.294,159.793
C01360=1017.873,250.239,-132.369,169.105,51.300,159.793
C01361=1017.867,249.990,-132.340,169.101,51.307,159.794
C01362=1017.861,249.742,-132.314,169.096,51.313,159.794
C01363=1017.856,249.513,-132.288,169.092,51.319,159.795
C01364=1017.851,249.286,-132.262,169.088,51.324,159.795
C01365=1017.845,249.058,-132.236,169.083,51.330,159.796
C01366=1017.840,248.829,-132.212,169.079,51.335,159.796
C01367=1017.835,248.601,-132.185,169.076,51.342,159.797
C01368=1017.828,248.372,-132.160,169.072,51.347,159.797
C01369=1017.823,248.144,-132.135,169.067,51.352,159.798
C01370=1017.818,247.915,-132.109,169.062,51.358,159.798
C01371=1017.812,247.668,-132.081,169.059,51.364,159.799
C01372=1017.807,247.419,-132.054,169.054,51.371,159.800
C01373=1017.800,247.170,-132.026,169.050,51.377,159.800
C01374=1017.795,246.922,-131.998,169.045,51.384,159.801
C01375=1017.789,246.673,-131.971,169.041,51.389,159.801
C01376=1017.783,246.425,-131.943,169.036,51.396,159.802
C01377=1017.777,246.177,-131.915,169.032,51.402,159.802
C01378=1017.772,245.928,-131.888,169.027,51.409,159.803
C01379=1017.766,245.680,-131.860,169.023,51.415,159.804
C01380=1017.760,245.431,-131.832,169.019,51.422,159.804
C01381=1017.755,245.183,-131.805,169.014,51.427,159.805
C01382=1017.749,244.935,-131.777,169.009,51.434,159.805
C01383=1017.744,244.686,-131.750,169.005,51.440,159.806
C01384=1017.737,244.438,-131.722,169.001,51.447,159.806
C01385=1017.732,244.190,-131.694,168.996,51.453,159.807
C01386=1017.726,243.940,-131.667,168.992,51.460,159.808
C01387=1017.720,243.693,-131.639,168.987,51.466,159.808
C01388=1017.715,243.444,-131.612,168.983,51.473,159.809
C01389=1017.709,243.196,-131.585,168.979,51.479,159.810
C01390=1017.704,242.947,-131.557,168.974,51.485,159.810
C01391=1017.698,242.699,-131.530,168.970,51.492,159.811
C01392=1017.691,242.450,-131.503,168.965,51.498,159.811
C01393=1017.686,242.201,-131.476,168.961,51.505,159.812
C01394=1017.680,241.954,-131.448,168.956,51.511,159.812
C01395=1017.674,241.705,-131.421,168.952,51.519,159.813
C01396=1017.668,241.457,-131.393,168.948,51.525,159.814
C01397=1017.663,241.208,-131.367,168.944,51.531,159.815
C01398=1017.657,240.960,-131.340,168.939,51.538,159.815
C01399=1017.651,240.710,-131.312,168.935,51.544,159.816
C01400=1017.645,240.463,-131.285,168.930,51.551,159.816
C01401=1017.639,240.214,-131.258,168.926,51.558,159.817
C01402=1017.634,239.966,-131.231,168.921,51.565,159.818
C01403=1017.628,239.717,-131.203,168.917,51.571,159.818
C01404=1017.622,239.469,-131.177,168.912,51.578,159.819
C01405=1017.617,239.220,-131.150,168.909,51.585,159.820
C01406=1017.611,238.972,-131.123,168.904,51.591,159.820
C01407=1017.605,238.723,-131.096,168.900,51.598,159.821
C01408=1017.599,238.475,-131.068,168.895,51.605,159.822
C01409=1017.593,238.227,-131.042,168.891,51.611,159.822
C01410=1017.587,237.978,-131.015,168.887,51.619,159.823
C01411=1017.581,237.730,-130.989,168.882,51.625,159.824
C01412=1017.575,237.481,-130.962,168.878,51.632,159.824
C01413=1017.569,237.233,-130.935,168.873,51.639,159.825
C01414=1017.563,236.984,-130.908,168.869,51.645,159.826
C01415=1017.558,236.736,-130.881,168.865,51.653,159.826
C01416=1017.553,236.487,-130.854,168.860,51.659,159.827
C01417=1017.546,236.238,-130.827,168.856,51.666,159.828
C01418=1017.540,235.990,-130.801,168.851,51.673,159.828
C01419=1017.535,235.741,-130.774,168.847,51.680,159.829
C01420=1017.529,235.493,-130.747,168.843,51.687,159.830
C01421=1017.523,235.245,-130.721,168.838,51.694,159.831
C01422=1017.517,234.996,-130.694,168.834,51.701,159.831
C01423=1017.512,234.765,-130.669,168.831,51.707,159.832
C01424=1017.506,234.533,-130.645,168.826,51.714,159.833
C01425=1017.500,234.301,-130.620,168.823,51.720,159.833
C01426=1017.495,234.070,-130.595,168.818,51.727,159.834
C01427=1017.490,233.838,-130.571,168.813,51.733,159.834
C01428=1017.485,233.607,-130.546,168.810,51.740,159.835
C01429=1017.479,233.374,-130.521,168.806,51.747,159.836
C01430=1017.474,233.143,-130.496,168.802,51.753,159.837
C01431=1017.467,232.895,-130.470,168.798,51.760,159.837
C01432=1017.462,232.646,-130.443,168.793,51.767,159.838
C01433=1017.456,232.397,-130.417,168.789,51.774,159.839
C01434=1017.450,232.149,-130.391,168.785,51.781,159.840
C01435=1017.445,231.901,-130.364,168.781,51.788,159.840
C01436=1017.439,231.652,-130.337,168.776,51.795,159.841
C01437=1017.433,231.404,-130.311,168.772,51.802,159.842
C01438=1017.427,231.155,-130.285,168.768,51.810,159.843
C01439=1017.422,230.907,-130.258,168.764,51.816,159.843
C01440=1017.416,230.658,-130.232,168.759,51.823,159.844
C01441=1017.410,230.409,-130.206,168.755,51.831,159.845
C01442=1017.405,230.161,-130.179,168.751,51.838,159.845
C01443=1017.399,229.913,-130.152,168.746,51.846,159.846
C01444=1017.393,229.664,-130.126,168.741,51.852,159.847
C01445=1017.388,229.415,-130.100,168.737,51.859,159.848
C01446=1017.382,229.167,-130.073,168.733,51.867,159.848
C01447=1017.376,228.918,-130.048,168.729,51.874,159.849
C01448=1017.370,228.670,-130.021,168.725,51.881,159.850
C01449=1017.364,228.421,-129.995,168.721,51.888,159.851
C01450=1017.359,228.172,-129.968,168.717,51.896,159.852
C01451=1017.353,227.923,-129.943,168.712,51.903,159.852
C01452=1017.347,227.675,-129.916,168.708,51.910,159.853
C01453=1017.341,227.427,-129.890,168.704,51.918,159.854
C01454=1017.335,227.178,-129.864,168.699,51.925,159.855
C01455=1017.330,226.930,-129.837,168.695,51.932,159.855
C01456=1017.324,226.681,-129.811,168.691,51.940,159.856
C01457=1017.319,226.432,-129.785,168.687,51.947,159.857
C01458=1017.312,226.184,-129.759,168.683,51.954,159.858
C01459=1017.307,225.935,-129.733,168.678,51.962,159.859
C01460=1017.300,225.687,-129.707,168.673,51.969,159.859
C01461=1017.295,225.438,-129.681,168.670,51.977,159.860
C01462=1017.289,225.189,-129.655,168.666,51.984,159.861
C01463=1017.284,224.941,-129.631,168.661,51.992,159.862
C01464=1017.278,224.692,-129.604,168.657,51.999,159.863
C01465=1017.272,224.444,-129.579,168.653,52.006,159.863
C01466=1017.266,224.195,-129.553,168.649,52.015,159.864
C01467=1017.260,223.947,-129.527,168.644,52.022,159.865
C01468=1017.254,223.698,-129.501,168.640,52.029,159.866
C01469=1017.249,223.449,-129.475,168.636,52.036,159.867
C01470=1017.243,223.200,-129.449,168.631,52.045,159.868
C01471=1017.237,222.952,-129.423,168.627,52.052,159.868
C01472=1017.231,222.704,-129.398,168.623,52.059,159.869
C01473=1017.226,222.455,-129.372,168.619,52.067,159.870
C01474=1017.220,222.206,-129.346,168.616,52.075,159.871
C01475=1017.214,221.957,-129.321,168.610,52.082,159.872
C01476=1017.209,221.708,-129.295,168.606,52.090,159.873
C01477=1017.202,221.460,-129.269,168.603,52.098,159.874
C01478=1017.197,221.212,-129.243,168.599,52.105,159.874
C01479=1017.191,220.963,-129.218,168.594,52.113,159.875
C01480=1017.186,220.714,-129.192,168.590,52.121,159.876
C01481=1017.179,220.465,-129.166,168.586,52.128,159.877
C01482=1017.174,220.216,-129.140,168.582,52.136,159.878
C01483=1017.169,219.981,-129.116,168.578,52.143,159.879
C01484=1017.163,219.745,-129.091,168.574,52.151,159.879
C01485=1017.158,219.510,-129.067,168.570,52.158,159.880
C01486=1017.153,219.274,-129.043,168.566,52.165,159.881
C01487=1017.147,219.039,-129.019,168.562,52.172,159.882
C01488=1017.142,218.803,-128.995,168.557,52.180,159.883
C01489=1017.136,218.567,-128.971,168.553,52.187,159.883
C01490=1017.131,218.331,-128.946,168.550,52.194,159.884
C01491=1017.125,218.082,-128.920,168.546,52.202,159.885
C01492=1017.120,217.834,-128.895,168.542,52.210,159.886
C01493=1017.114,217.585,-128.870,168.538,52.218,159.887
C01494=1017.107,217.337,-128.845,168.533,52.226,159.888
C01495=1017.102,217.088,-128.819,168.529,52.233,159.889
C01496=1017.096,216.840,-128.794,168.526,52.241,159.890
C01497=1017.090,216.591,-128.768,168.521,52.250,159.891
C01498=1017.085,216.341,-128.743,168.517,52.257,159.891
C01499=1017.079,216.093,-128.718,168.512,52.266,159.892
C01500=1017.073,215.845,-128.693,168.509,52.274,159.893
C01501=1017.067,215.596,-128.668,168.504,52.281,159.894
C01502=1017.061,215.347,-128.642,168.500,52.289,159.895
C01503=1017.056,215.099,-128.617,168.496,52.297,159.896
C01504=1017.050,214.850,-128.592,168.491,52.306,159.897
C01505=1017.044,214.601,-128.567,168.488,52.314,159.898
C01506=1017.039,214.353,-128.541,168.484,52.321,159.899
C01507=1017.033,214.104,-128.517,168.479,52.329,159.900
C01508=1017.027,213.855,-128.491,168.476,52.337,159.901
C01509=1017.021,213.607,-128.466,168.471,52.346,159.902
C01510=1017.016,213.358,-128.440,168.467,52.354,159.903
C01511=1017.010,213.109,-128.416,168.463,52.361,159.903
C01512=1017.004,212.861,-128.391,168.459,52.370,159.904
C01513=1016.998,212.612,-128.365,168.455,52.378,159.905
C01514=1016.993,212.363,-128.341,168.450,52.386,159.906
C01515=1016.987,212.115,-128.315,168.447,52.394,159.907
C01516=1016.981,211.866,-128.290,168.443,52.402,159.908
C01517=1016.976,211.617,-128.266,168.438,52.411,159.909
C01518=1016.970,211.368,-128.240,168.435,52.419,159.910
C01519=1016.965,211.120,-128.215,168.430,52.427,159.911
C01520=1016.959,210.871,-128.190,168.427,52.435,159.912
C01521=1016.953,210.622,-128.165,168.422,52.443,159.913
C01522=1016.948,210.374,-128.140,168.418,52.451,159.914
C01523=1016.942,210.125,-128.115,168.413,52.459,159.915
C01524=1016.936,209.877,-128.090,168.410,52.467,159.916
C01525=1016.930,209.628,-128.065,168.405,52.476,159.917
C01526=1016.925,209.380,-128.040,168.402,52.484,159.918
C01527=1016.920,209.130,-128.015,168.397,52.493,159.919
C01528=1016.914,208.882,-127.990,168.394,52.501,159.920
C01529=1016.908,208.633,-127.965,168.389,52.509,159.921
C01530=1016.903,208.384,-127.941,168.386,52.517,159.922
C01531=1016.896,208.136,-127.916,168.381,52.526,159.923
C01532=1016.891,207.887,-127.891,168.377,52.534,159.924
C01533=1016.885,207.638,-127.866,168.373,52.542,159.925
C01534=1016.880,207.390,-127.842,168.370,52.551,159.926
C01535=1016.873,207.141,-127.816,168.365,52.560,159.927
C01536=1016.868,206.892,-127.792,168.361,52.568,159.928
C01537=1016.862,206.643,-127.767,168.357,52.576,159.929
C01538=1016.857,206.395,-127.743,168.353,52.585,159.930
C01539=1016.851,206.146,-127.718,168.349,52.593,159.931
C01540=1016.845,205.897,-127.694,168.344,52.602,159.932
C01541=1016.839,205.649,-127.668,168.341,52.610,159.933
C01542=1016.834,205.400,-127.644,168.337,52.619,159.934
C01543=1016.828,205.161,-127.620,168.333,52.627,159.935
C01544=1016.823,204.924,-127.597,168.329,52.635,159.936
C01545=1016.817,204.685,-127.574,168.325,52.643,159.937
C01546=1016.812,204.447,-127.550,168.321,52.652,159.938
C01547=1016.806,204.209,-127.527,168.317,52.660,159.939
C01548=1016.800,203.971,-127.504,168.313,52.668,159.940
C01549=1016.795,203.733,-127.480,168.310,52.676,159.941
C01550=1016.770,202.498,-127.365,167.815,52.600,159.826
C01551=1016.766,202.249,-127.342,167.810,52.611,159.827
C01552=1016.762,202.000,-127.320,167.805,52.620,159.828
C01553=1016.757,201.752,-127.297,167.801,52.630,159.829
C01554=1016.752,201.503,-127.274,167.796,52.640,159.830
C01555=1016.747,201.254,-127.252,167.791,52.650,159.831
C01556=1016.742,201.006,-127.229,167.787,52.659,159.832
C01557=1016.738,200.756,-127.206,167.782,52.669,159.833
C01558=1016.733,200.508,-127.183,167.777,52.679,159.834
C01559=1016.729,200.258,-127.161,167.773,52.689,159.836
C01560=1016.724,200.010,-127.137,167.768,52.698,159.836
C01561=1016.719,199.760,-127.115,167.764,52.708,159.838
C01562=1016.714,199.512,-127.092,167.759,52.718,159.839
C01563=1016.710,199.263,-127.070,167.754,52.728,159.840
C01564=1016.705,199.013,-127.047,167.750,52.737,159.841
C01565=1016.700,198.765,-127.024,167.745,52.747,159.842
C01566=1016.696,198.516,-127.002,167.741,52.758,159.843
C01567=1016.690,198.266,-126.980,167.736,52.767,159.844
C01568=1016.686,198.018,-126.957,167.732,52.777,159.845
C01569=1016.681,197.769,-126.935,167.727,52.787,159.847
C01570=1016.676,197.520,-126.913,167.722,52.798,159.848
C01571=1016.671,197.270,-126.890,167.718,52.807,159.849
C01572=1016.667,197.022,-126.869,167.713,52.817,159.850
C01573=1016.661,196.773,-126.846,167.708,52.827,159.851
C01574=1016.657,196.525,-126.824,167.704,52.837,159.852
C01575=1016.652,196.275,-126.801,167.699,52.847,159.853
C01576=1016.647,196.026,-126.779,167.695,52.857,159.855
C01577=1016.642,195.777,-126.758,167.691,52.867,159.856
C01578=1016.638,195.528,-126.735,167.686,52.877,159.857
C01579=1016.633,195.280,-126.712,167.681,52.887,159.858
C01580=1016.628,195.030,-126.690,167.677,52.897,159.859
C01581=1016.623,194.781,-126.668,167.672,52.907,159.860
C01582=1016.619,194.532,-126.646,167.668,52.916,159.861
C01583=1016.614,194.284,-126.624,167.664,52.927,159.863
C01584=1016.609,194.035,-126.602,167.659,52.937,159.864
C01585=1016.605,193.786,-126.580,167.655,52.946,159.865
C01586=1016.600,193.536,-126.558,167.650,52.957,159.866
C01587=1016.595,193.287,-126.536,167.646,52.967,159.867
C01588=1016.591,193.038,-126.513,167.642,52.977,159.868
C01589=1016.586,192.789,-126.491,167.636,52.986,159.869
C01590=1016.581,192.541,-126.469,167.633,52.996,159.871
C01591=1016.576,192.292,-126.448,167.628,53.007,159.872
C01592=1016.572,192.043,-126.425,167.624,53.017,159.873
C01593=1016.567,191.793,-126.403,167.619,53.026,159.874
C01594=1016.562,191.544,-126.381,167.614,53.037,159.875
C01595=1016.558,191.295,-126.359,167.611,53.047,159.877
C01596=1016.553,191.046,-126.337,167.606,53.056,159.877
C01597=1016.548,190.797,-126.315,167.602,53.066,159.879
C01598=1016.543,190.549,-126.293,167.597,53.077,159.880
C01599=1016.539,190.300,-126.271,167.593,53.086,159.881
C01600=1016.534,190.051,-126.249,167.588,53.096,159.882
C01601=1016.530,189.802,-126.227,167.585,53.106,159.883
C01602=1016.526,189.553,-126.204,167.580,53.116,159.885
C01603=1016.521,189.304,-126.182,167.576,53.126,159.886
C01604=1016.516,189.055,-126.161,167.571,53.136,159.887
C01605=1016.511,188.806,-126.139,167.567,53.146,159.888
C01606=1016.507,188.557,-126.117,167.563,53.156,159.889
C01607=1016.502,188.308,-126.095,167.559,53.166,159.890
C01608=1016.498,188.059,-126.073,167.554,53.176,159.891
C01609=1016.493,187.810,-126.051,167.550,53.186,159.893
C01610=1016.489,187.561,-126.029,167.546,53.196,159.894
C01611=1016.483,187.280,-126.005,167.541,53.207,159.895
C01612=1016.478,187.001,-125.980,167.536,53.218,159.896
C01613=1016.473,186.720,-125.955,167.532,53.229,159.898
C01614=1016.468,186.440,-125.931,167.526,53.241,159.899
C01615=1016.463,186.191,-125.909,167.523,53.251,159.900
C01616=1016.459,185.942,-125.887,167.518,53.261,159.901
C01617=1016.454,185.693,-125.865,167.514,53.270,159.903
C01618=1016.450,185.445,-125.843,167.509,53.281,159.904
C01619=1016.445,185.195,-125.822,167.506,53.291,159.905
C01620=1016.441,184.946,-125.799,167.501,53.301,159.906
C01621=1016.436,184.697,-125.778,167.497,53.310,159.907
C01622=1016.432,184.448,-125.756,167.493,53.320,159.909
C01623=1016.427,184.200,-125.735,167.489,53.331,159.910
C01624=1016.423,183.951,-125.712,167.484,53.340,159.911
C01625=1016.419,183.702,-125.691,167.480,53.351,159.912
C01626=1016.414,183.452,-125.669,167.476,53.361,159.913
C01627=1016.410,183.203,-125.647,167.473,53.371,159.914
C01628=1016.405,182.954,-125.625,167.468,53.380,159.915
C01629=1016.401,182.705,-125.604,167.464,53.390,159.917
C01630=1016.396,182.456,-125.582,167.459,53.401,159.918
C01631=1016.392,182.206,-125.560,167.455,53.410,159.919
C01632=1016.387,181.957,-125.538,167.452,53.420,159.920
C01633=1016.383,181.709,-125.518,167.447,53.430,159.921
C01634=1016.378,181.460,-125.496,167.443,53.440,159.923
C01635=1016.373,181.211,-125.475,167.439,53.451,159.924
C01636=1016.369,180.961,-125.454,167.435,53.461,159.925
C01637=1016.364,180.713,-125.432,167.431,53.471,159.926
C01638=1016.359,180.463,-125.412,167.427,53.481,159.928
C01639=1016.354,180.214,-125.391,167.422,53.492,159.929
C01640=1016.350,179.965,-125.369,167.418,53.502,159.930
C01641=1016.345,179.717,-125.349,167.414,53.512,159.931
C01642=1016.340,179.467,-125.327,167.410,53.523,159.932
C01643=1016.335,179.218,-125.307,167.406,53.533,159.934
C01644=1016.330,178.969,-125.286,167.401,53.543,159.935
C01645=1016.326,178.719,-125.265,167.398,53.553,159.936
C01646=1016.320,178.471,-125.243,167.393,53.564,159.937
C01647=1016.316,178.222,-125.222,167.390,53.574,159.939
C01648=1016.312,177.973,-125.201,167.386,53.585,159.940
C01649=1016.307,177.724,-125.181,167.382,53.595,159.941
C01650=1016.302,177.474,-125.160,167.377,53.605,159.943
C01651=1016.297,177.225,-125.139,167.374,53.615,159.944
C01652=1016.293,176.977,-125.118,167.369,53.626,159.945
C01653=1016.288,176.727,-125.096,167.366,53.636,159.946
C01654=1016.283,176.478,-125.076,167.361,53.646,159.947
C01655=1016.278,176.229,-125.055,167.358,53.657,159.949
C01656=1016.273,175.980,-125.034,167.353,53.667,159.950
C01657=1016.269,175.731,-125.013,167.350,53.677,159.951
C01658=1016.265,175.482,-124.992,167.345,53.688,159.952
C01659=1016.259,175.232,-124.972,167.341,53.698,159.954
C01660=1016.255,174.983,-124.951,167.337,53.708,159.955
C01661=1016.250,174.735,-124.930,167.333,53.718,159.956
C01662=1016.245,174.486,-124.908,167.330,53.728,159.957
C01663=1016.241,174.236,-124.887,167.325,53.739,159.959
C01664=1016.236,173.988,-124.867,167.322,53.749,159.960
C01665=1016.232,173.739,-124.846,167.317,53.759,159.961
C01666=1016.226,173.489,-124.825,167.314,53.769,159.962
C01667=1016.222,173.241,-124.805,167.309,53.780,159.964
C01668=1016.218,172.991,-124.784,167.306,53.790,159.965
C01669=1016.213,172.742,-124.763,167.302,53.800,159.966
C01670=1016.208,172.493,-124.742,167.298,53.811,159.967
C01671=1016.204,172.244,-124.721,167.294,53.821,159.969
C01672=1016.199,171.995,-124.700,167.290,53.831,159.970
C01673=1016.195,171.746,-124.680,167.286,53.841,159.971
C01674=1016.190,171.496,-124.660,167.283,53.851,159.972
C01675=1016.185,171.216,-124.636,167.277,53.863,159.974
C01676=1016.180,170.935,-124.612,167.274,53.875,159.975
C01677=1016.175,170.655,-124.590,167.269,53.886,159.977
C01678=1016.170,170.375,-124.566,167.265,53.898,159.978
C01679=1016.164,170.126,-124.545,167.261,53.908,159.979
C01680=1016.161,169.876,-124.525,167.257,53.918,159.981
C01681=1016.156,169.627,-124.504,167.253,53.928,159.982
C01682=1016.151,169.378,-124.483,167.250,53.939,159.983
C01683=1016.147,169.129,-124.463,167.245,53.949,159.984
C01684=1016.142,168.880,-124.442,167.242,53.959,159.986
C01685=1016.138,168.631,-124.421,167.238,53.969,159.987
C01686=1016.133,168.382,-124.400,167.234,53.980,159.988
C01687=1016.128,168.132,-124.380,167.230,53.990,159.989
C01688=1016.125,167.883,-124.359,167.227,54.000,159.991
C01689=1016.119,167.634,-124.339,167.222,54.011,159.992
C01690=1016.115,167.385,-124.318,167.219,54.021,159.993
C01691=1016.111,167.136,-124.297,167.216,54.031,159.995
C01692=1016.106,166.888,-124.277,167.211,54.042,159.996
C01693=1016.102,166.638,-124.256,167.208,54.052,159.997
C01694=1016.097,166.389,-124.236,167.204,54.062,159.998
C01695=1016.093,166.140,-124.215,167.201,54.072,160.000
C01696=1016.089,165.891,-124.194,167.196,54.083,160.001
C01697=1016.084,165.641,-124.174,167.192,54.092,160.002
C01698=1016.080,165.392,-124.154,167.189,54.102,160.003
C01699=1016.075,165.143,-124.133,167.185,54.112,160.005
C01700=1016.071,164.895,-124.112,167.181,54.123,160.006
C01701=1016.066,164.645,-124.092,167.178,54.133,160.007
C01702=1016.062,164.396,-124.072,167.174,54.143,160.008
C01703=1016.058,164.147,-124.050,167.171,54.153,160.010
C01704=1016.053,163.898,-124.030,167.166,54.164,160.011
C01705=1016.049,163.648,-124.010,167.163,54.174,160.012
C01706=1016.044,163.400,-123.990,167.159,54.184,160.013
C01707=1016.039,163.150,-123.969,167.156,54.194,160.015
C01708=1016.036,162.901,-123.948,167.152,54.205,160.016
C01709=1016.031,162.652,-123.928,167.148,54.215,160.017
C01710=1016.027,162.403,-123.907,167.145,54.225,160.019
C01711=1016.022,162.153,-123.887,167.141,54.235,160.020
C01712=1016.018,161.905,-123.867,167.137,54.245,160.021
C01713=1016.013,161.656,-123.846,167.133,54.256,160.022
C01714=1016.009,161.406,-123.826,167.130,54.266,160.023
C01715=1016.005,161.157,-123.805,167.126,54.276,160.025
C01716=1016.000,160.908,-123.785,167.123,54.286,160.026
C01717=1015.996,160.659,-123.764,167.119,54.296,160.027
C01718=1015.992,160.411,-123.744,167.116,54.307,160.029
C01719=1015.987,160.161,-123.724,167.112,54.317,160.030
C01720=1015.983,159.912,-123.704,167.108,54.327,160.031
C01721=1015.978,159.662,-123.683,167.104,54.337,160.032
C01722=1015.975,159.413,-123.662,167.101,54.347,160.034
C01723=1015.970,159.164,-123.643,167.098,54.357,160.035
C01724=1015.966,158.915,-123.622,167.094,54.368,160.036
C01725=1015.961,158.666,-123.602,167.091,54.378,160.038
C01726=1015.957,158.417,-123.582,167.088,54.388,160.039
C01727=1015.952,158.167,-123.562,167.083,54.399,160.040
C01728=1015.948,157.919,-123.542,167.080,54.409,160.041
C01729=1015.943,157.669,-123.522,167.076,54.419,160.043
C01730=1015.938,157.420,-123.502,167.072,54.430,160.044
C01731=1015.934,157.172,-123.482,167.069,54.440,160.045
C01732=1015.930,156.922,-123.462,167.066,54.451,160.047
C01733=1015.925,156.673,-123.442,167.062,54.461,160.048
C01734=1015.921,156.424,-123.423,167.058,54.472,160.049
C01735=1015.916,156.174,-123.402,167.055,54.482,160.051
C01736=1015.911,155.925,-123.383,167.051,54.492,160.052
C01737=1015.907,155.676,-123.363,167.048,54.502,160.053
C01738=1015.902,155.427,-123.343,167.044,54.513,160.054
C01739=1015.897,155.146,-123.321,167.040,54.525,160.056
C01740=1015.892,154.865,-123.299,167.036,54.536,160.058
C01741=1015.887,154.584,-123.276,167.032,54.548,160.059
C01742=1015.882,154.304,-123.254,167.028,54.560,160.061
C01743=1015.878,154.055,-123.234,167.025,54.570,160.062
C01744=1015.873,153.806,-123.215,167.022,54.581,160.063
C01745=1015.868,153.556,-123.195,167.018,54.591,160.065
C01746=1015.864,153.307,-123.175,167.014,54.602,160.066
C01747=1015.859,153.059,-123.155,167.011,54.612,160.067
C01748=1015.854,152.809,-123.135,167.007,54.622,160.068
C01749=1015.850,152.560,-123.116,167.004,54.632,160.070
C01750=1015.846,152.311,-123.096,167.001,54.643,160.071
C01751=1015.841,152.062,-123.077,166.996,54.653,160.072
C01752=1015.836,151.812,-123.057,166.994,54.664,160.074
C01753=1015.832,151.563,-123.038,166.990,54.675,160.075
C01754=1015.828,151.314,-123.018,166.987,54.685,160.076
C01755=1015.823,151.065,-122.999,166.983,54.696,160.078
C01756=1015.818,150.815,-122.979,166.979,54.706,160.079
C01757=1015.814,150.566,-122.959,166.976,54.716,160.080
C01758=1015.810,150.317,-122.940,166.973,54.726,160.082
C01759=1015.805,150.068,-122.920,166.969,54.737,160.083
C01760=1015.800,149.818,-122.901,166.965,54.747,160.084
C01761=1015.796,149.569,-122.881,166.962,54.758,160.086
C01762=1015.792,149.320,-122.862,166.959,54.769,160.087
C01763=1015.787,149.071,-122.842,166.956,54.779,160.088
C01764=1015.783,148.822,-122.823,166.953,54.789,160.090
C01765=1015.778,148.572,-122.803,166.948,54.800,160.091
C01766=1015.773,148.324,-122.784,166.945,54.810,160.092
C01767=1015.769,148.075,-122.764,166.942,54.820,160.094
C01768=1015.765,147.825,-122.746,166.938,54.831,160.095
C01769=1015.760,147.576,-122.726,166.935,54.841,160.096
C01770=1015.755,147.326,-122.706,166.932,54.851,160.098
C01771=1015.751,147.077,-122.687,166.928,54.863,160.099
C01772=1015.747,146.828,-122.667,166.925,54.873,160.100
C01773=1015.742,146.579,-122.648,166.922,54.883,160.102
C01774=1015.738,146.330,-122.629,166.918,54.894,160.103
C01775=1015.733,146.081,-122.610,166.915,54.904,160.104
C01776=1015.728,145.831,-122.591,166.912,54.914,160.106
C01777=1015.724,145.582,-122.571,166.909,54.925,160.107
